LIN {X 0,Y 338.105,Z 590.455,A -85,B 0,C 180,E1 14436.471,E2 14436.471} C_VEL
LIN {X 0,Y 336.895,Z 591.514,A -85,B 0,C 180,E1 14436.227,E2 14436.227} C_VEL
LIN {X 0,Y 331.702,Z 598.648,A -85,B 0,C 180,E1 14435.239,E2 14435.239} C_VEL
LIN {X 0,Y 327.518,Z 602.639,A -85,B 0,C 180,E1 14434.334,E2 14434.334} C_VEL
LIN {X 0,Y 325.57,Z 603.97,A -85,B 0,C 180,E1 14433.877,E2 14433.877} C_VEL
LIN {X 0,Y 320.508,Z 612.012,A -85,B 0,C 180,E1 14432.822,E2 14432.822} C_VEL
LIN {X 0,Y 316.738,Z 616.286,A -85,B 0,C 180,E1 14431.922,E2 14431.922} C_VEL
LIN {X 0,Y 314.815,Z 617.214,A -85,B 0,C 180,E1 14431.391,E2 14431.391} C_VEL
LIN {X 0,Y 314.423,Z 617.302,A -85,B 0,C 180,E1 14431.251,E2 14431.251} C_VEL
LIN {X 0,Y 311.704,Z 638.432,A -85,B 0,C 180,E1 14428.545,E2 14428.545} C_VEL
LIN {X 0,Y 311.765,Z 644.155,A -85,B 0,C 180,E1 14428.291,E2 14428.291} C_VEL
LIN {X 0,Y 303.31,Z 754.586,A -85,B 0,C 180,E1 14423.992,E2 14423.992} C_VEL
LIN {X 0,Y 301.747,Z 787.034,A -85,B 0,C 180,E1 14422.515,E2 14422.515} C_VEL
LIN {X 0,Y 300.704,Z 803.184,A -85,B 0,C 180,E1 14421.454,E2 14421.454} C_VEL
LIN {X 0,Y 299.299,Z 819.779,A -85,B 0,C 180,E1 14419.987,E2 14419.987} C_VEL
LIN {X 0,Y 297.78,Z 834.708,A -85,B 0,C 180,E1 14418.298,E2 14418.298} C_VEL
LIN {X 0,Y 296.083,Z 849.627,A -85,B 0,C 180,E1 14416.177,E2 14416.177} C_VEL
LIN {X 0,Y 294.448,Z 863.222,A -85,B 0,C 180,E1 14413.751,E2 14413.751} C_VEL
LIN {X 0,Y 293.091,Z 874.714,A -85,B 0,C 180,E1 14411.213,E2 14411.213} C_VEL
LIN {X 0,Y 291.948,Z 885.373,A -85,B 0,C 180,E1 14408.27,E2 14408.27} C_VEL
LIN {X 0,Y 291.167,Z 894.27,A -85,B 0,C 180,E1 14405.123,E2 14405.123} C_VEL
LIN {X 0,Y 290.847,Z 900.711,A -85,B 0,C 180,E1 14402.167,E2 14402.167} C_VEL
LIN {X 0,Y 290.9,Z 906.041,A -85,B 0,C 180,E1 14398.819,E2 14398.819} C_VEL
LIN {X 0,Y 291.395,Z 909.402,A -85,B 0,C 180,E1 14395.474,E2 14395.474} C_VEL
LIN {X 0,Y 292.318,Z 910.935,A -85,B 0,C 180,E1 14392.334,E2 14392.334} C_VEL
LIN {X 0,Y 293.979,Z 910.74,A -85,B 0,C 180,E1 14388.822,E2 14388.822} C_VEL
LIN {X 0,Y 296.38,Z 908.513,A -85,B 0,C 180,E1 14385.344,E2 14385.344} C_VEL
LIN {X 0,Y 299.304,Z 904.667,A -85,B 0,C 180,E1 14382.193,E2 14382.193} C_VEL
LIN {X 0,Y 302.949,Z 899.041,A -85,B 0,C 180,E1 14379.118,E2 14379.118} C_VEL
LIN {X 0,Y 307.224,Z 891.662,A -85,B 0,C 180,E1 14376.2,E2 14376.2} C_VEL
LIN {X 0,Y 311.889,Z 882.811,A -85,B 0,C 180,E1 14373.538,E2 14373.538} C_VEL
LIN {X 0,Y 317.212,Z 871.822,A -85,B 0,C 180,E1 14370.961,E2 14370.961} C_VEL
LIN {X 0,Y 322.811,Z 859.287,A -85,B 0,C 180,E1 14368.644,E2 14368.644} C_VEL
LIN {X 0,Y 328.898,Z 844.76,A -85,B 0,C 180,E1 14366.512,E2 14366.512} C_VEL
LIN {X 0,Y 335.235,Z 828.569,A -85,B 0,C 180,E1 14364.647,E2 14364.647} C_VEL
LIN {X 0,Y 344.132,Z 807.464,A -85,B 0,C 180,E1 14362.715,E2 14362.715} C_VEL
LIN {X 0,Y 354.941,Z 783.665,A -85,B 0,C 180,E1 14360.98,E2 14360.98} C_VEL
LIN {X 0,Y 365.49,Z 758.939,A -85,B 0,C 180,E1 14359.583,E2 14359.583} C_VEL
LIN {X 0,Y 366.222,Z 757.158,A -85,B 0,C 180,E1 14359.481,E2 14359.481} C_VEL
LIN {X 0,Y 359.783,Z 774.746,A -85,B 0,C 180,E1 14358.984,E2 14358.984} C_VEL
LIN {X 0,Y 353.257,Z 791.701,A -85,B 0,C 180,E1 14358.23,E2 14358.23} C_VEL
LIN {X 0,Y 342.525,Z 818.157,A -85,B 0,C 180,E1 14356.624,E2 14356.624} C_VEL
LIN {X 0,Y 334.303,Z 838.121,A -85,B 0,C 180,E1 14355.081,E2 14355.081} C_VEL
LIN {X 0,Y 330.317,Z 857.082,A -85,B 0,C 180,E1 14353.883,E2 14353.883} C_VEL
LIN {X 0,Y 325.728,Z 875.895,A -85,B 0,C 180,E1 14352.361,E2 14352.361} C_VEL
LIN {X 0,Y 320.539,Z 894.611,A -85,B 0,C 180,E1 14350.454,E2 14350.454} C_VEL
LIN {X 0,Y 315.4,Z 911.334,A -85,B 0,C 180,E1 14348.35,E2 14348.35} C_VEL
LIN {X 0,Y 310.233,Z 927.162,A -85,B 0,C 180,E1 14345.915,E2 14345.915} C_VEL
LIN {X 0,Y 305.231,Z 941.839,A -85,B 0,C 180,E1 14343.166,E2 14343.166} C_VEL
LIN {X 0,Y 300.629,Z 955.074,A -85,B 0,C 180,E1 14340.147,E2 14340.147} C_VEL
LIN {X 0,Y 296.615,Z 966.984,A -85,B 0,C 180,E1 14336.854,E2 14336.854} C_VEL
LIN {X 0,Y 293.159,Z 978.066,A -85,B 0,C 180,E1 14333.094,E2 14333.094} C_VEL
LIN {X 0,Y 290.587,Z 987.507,A -85,B 0,C 180,E1 14329.081,E2 14329.081} C_VEL
LIN {X 0,Y 289.081,Z 994.669,A -85,B 0,C 180,E1 14325.207,E2 14325.207} C_VEL
LIN {X 0,Y 288.342,Z 1000.295,A -85,B 0,C 180,E1 14321.198,E2 14321.198} C_VEL
LIN {X 0,Y 288.162,Z 1003.977,A -85,B 0,C 180,E1 14317.377,E2 14317.377} C_VEL
LIN {X 0,Y 288.251,Z 1006.151,A -85,B 0,C 180,E1 14313.581,E2 14313.581} C_VEL
LIN {X 0,Y 288.329,Z 1006.883,A -85,B 0,C 180,E1 14310.001,E2 14310.001} C_VEL
LIN {X 0,Y 288.247,Z 1006.145,A -85,B 0,C 180,E1 14306.421,E2 14306.421} C_VEL
LIN {X 0,Y 288.144,Z 1003.964,A -85,B 0,C 180,E1 14302.625,E2 14302.625} C_VEL
LIN {X 0,Y 288.325,Z 1000.281,A -85,B 0,C 180,E1 14298.803,E2 14298.803} C_VEL
LIN {X 0,Y 289.07,Z 994.6,A -85,B 0,C 180,E1 14294.76,E2 14294.76} C_VEL
LIN {X 0,Y 290.554,Z 987.48,A -85,B 0,C 180,E1 14290.919,E2 14290.919} C_VEL
LIN {X 0,Y 292.964,Z 978.552,A -85,B 0,C 180,E1 14287.104,E2 14287.104} C_VEL
LIN {X 0,Y 296.275,Z 967.843,A -85,B 0,C 180,E1 14283.42,E2 14283.42} C_VEL
LIN {X 0,Y 300.323,Z 955.793,A -85,B 0,C 180,E1 14280.041,E2 14280.041} C_VEL
LIN {X 0,Y 304.862,Z 942.662,A -85,B 0,C 180,E1 14277.015,E2 14277.015} C_VEL
LIN {X 0,Y 309.992,Z 927.6,A -85,B 0,C 180,E1 14274.173,E2 14274.173} C_VEL
LIN {X 0,Y 315.053,Z 912.094,A -85,B 0,C 180,E1 14271.769,E2 14271.769} C_VEL
LIN {X 0,Y 320.25,Z 895.206,A -85,B 0,C 180,E1 14269.622,E2 14269.622} C_VEL
LIN {X 0,Y 325.17,Z 877.603,A -85,B 0,C 180,E1 14267.802,E2 14267.802} C_VEL
LIN {X 0,Y 329.756,Z 859.099,A -85,B 0,C 180,E1 14266.266,E2 14266.266} C_VEL
LIN {X 0,Y 333.969,Z 839.227,A -85,B 0,C 180,E1 14264.985,E2 14264.985} C_VEL
LIN {X 0,Y 337.417,Z 818.867,A -85,B 0,C 180,E1 14264.011,E2 14264.011} C_VEL
LIN {X 0,Y 339.946,Z 798.236,A -85,B 0,C 180,E1 14263.309,E2 14263.309} C_VEL
LIN {X 0,Y 341.701,Z 774.328,A -85,B 0,C 180,E1 14262.775,E2 14262.775} C_VEL
LIN {X 0,Y 344.693,Z 746.04,A -85,B 0,C 180,E1 14262.462,E2 14262.462} C_VEL
LIN {X 0,Y 348.273,Z 722.638,A -85,B 0,C 180,E1 14262.405,E2 14262.405} C_VEL
LIN {X 0,Y 349.346,Z 716.122,A -85,B 0,C 180,E1 14262.403,E2 14262.403} C_VEL
LIN {X 0,Y 343.198,Z 700.036,A -85,B 0,C 180,E1 14260.778,E2 14260.778} C_VEL
LIN {X 0,Y 338.934,Z 686.753,A -85,B 0,C 180,E1 14259.515,E2 14259.515} C_VEL
LIN {X 0,Y 337.267,Z 665.975,A -85,B 0,C 180,E1 14256.787,E2 14256.787} C_VEL
LIN {X 0,Y 338.08,Z 643.412,A -85,B 0,C 180,E1 14253.984,E2 14253.984} C_VEL
LIN {X 0,Y 341.699,Z 617.006,A -85,B 0,C 180,E1 14250.98,E2 14250.98} C_VEL
LIN {X 0,Y 346.458,Z 593.984,A -85,B 0,C 180,E1 14248.53,E2 14248.53} C_VEL
LIN {X 0,Y 338.453,Z 575.878,A -85,B 0,C 180,E1 14244.616,E2 14244.616} C_VEL
LIN {X 0,Y 330.252,Z 558.135,A -85,B 0,C 180,E1 14240.375,E2 14240.375} C_VEL
LIN {X 0,Y 322.963,Z 542.982,A -85,B 0,C 180,E1 14236.363,E2 14236.363} C_VEL
LIN {X 0,Y 316.245,Z 529.387,A -85,B 0,C 180,E1 14232.415,E2 14232.415} C_VEL
LIN {X 0,Y 309.793,Z 516.677,A -85,B 0,C 180,E1 14228.351,E2 14228.351} C_VEL
LIN {X 0,Y 304.602,Z 506.811,A -85,B 0,C 180,E1 14224.896,E2 14224.896} C_VEL
LIN {X 0,Y 301.925,Z 501.833,A -85,B 0,C 180,E1 14223.037,E2 14223.037} C_VEL
LIN {X 0,Y 299.876,Z 497.861,A -85,B 0,C 180,E1 14221.528,E2 14221.528} C_VEL
LIN {X 0,Y 297.644,Z 493.478,A -85,B 0,C 180,E1 14219.807,E2 14219.807} C_VEL
LIN {X 0,Y 295.15,Z 488.762,A -85,B 0,C 180,E1 14217.864,E2 14217.864} C_VEL
LIN {X 0,Y 293.163,Z 485.098,A -85,B 0,C 180,E1 14216.284,E2 14216.284} C_VEL
LIN {X 0,Y 292.668,Z 484.054,A -85,B 0,C 180,E1 14215.797,E2 14215.797} C_VEL
LIN {X 0,Y 295.376,Z 485.784,A -85,B 0,C 180,E1 14210.452,E2 14210.452} C_VEL
LIN {X 0,Y 296.859,Z 489.544,A -85,B 0,C 180,E1 14207.617,E2 14207.617} C_VEL
LIN {X 0,Y 299.685,Z 492.227,A -85,B 0,C 180,E1 14204.519,E2 14204.519} C_VEL
LIN {X 0,Y 301.439,Z 495.849,A -85,B 0,C 180,E1 14202.431,E2 14202.431} C_VEL
LIN {X 0,Y 303.501,Z 497.912,A -85,B 0,C 180,E1 14200.765,E2 14200.765} C_VEL
LIN {X 0,Y 305.517,Z 501.787,A -85,B 0,C 180,E1 14198.859,E2 14198.859} C_VEL
LIN {X 0,Y 307.211,Z 503.912,A -85,B 0,C 180,E1 14197.617,E2 14197.617} C_VEL
LIN {X 0,Y 309.597,Z 507.894,A -85,B 0,C 180,E1 14195.785,E2 14195.785} C_VEL
LIN {X 0,Y 310.833,Z 509.839,A -85,B 0,C 180,E1 14194.976,E2 14194.976} C_VEL
LIN {X 0,Y 315.313,Z 515.527,A -85,B 0,C 180,E1 14192.983,E2 14192.983} C_VEL
LIN {X 0,Y 322.031,Z 524.183,A -85,B 0,C 180,E1 14190.315,E2 14190.315} C_VEL
LIN {X 0,Y 329.717,Z 535.071,A -85,B 0,C 180,E1 14187.589,E2 14187.589} C_VEL
LIN {X 0,Y 338.579,Z 548.442,A -85,B 0,C 180,E1 14184.788,E2 14184.788} C_VEL
LIN {X 0,Y 347.19,Z 562.872,A -85,B 0,C 180,E1 14182.32,E2 14182.32} C_VEL
LIN {X 0,Y 352.785,Z 573.372,A -85,B 0,C 180,E1 14180.813,E2 14180.813} C_VEL
LIN {X 0,Y 342.08,Z 768.353,A -85,B 0,C 180,E1 14176.743,E2 14176.743} C_VEL
LIN {X 0,Y 340.044,Z 788.682,A -85,B 0,C 180,E1 14176.065,E2 14176.065} C_VEL
LIN {X 0,Y 337.064,Z 809.308,A -85,B 0,C 180,E1 14175.089,E2 14175.089} C_VEL
LIN {X 0,Y 333.401,Z 828.945,A -85,B 0,C 180,E1 14173.848,E2 14173.848} C_VEL
LIN {X 0,Y 329.276,Z 847.192,A -85,B 0,C 180,E1 14172.384,E2 14172.384} C_VEL
LIN {X 0,Y 324.469,Z 865.449,A -85,B 0,C 180,E1 14170.556,E2 14170.556} C_VEL
LIN {X 0,Y 319.337,Z 882.593,A -85,B 0,C 180,E1 14168.425,E2 14168.425} C_VEL
LIN {X 0,Y 314.214,Z 898.139,A -85,B 0,C 180,E1 14166.063,E2 14166.063} C_VEL
LIN {X 0,Y 309.078,Z 912.768,A -85,B 0,C 180,E1 14163.362,E2 14163.362} C_VEL
LIN {X 0,Y 304.251,Z 925.958,A -85,B 0,C 180,E1 14160.403,E2 14160.403} C_VEL
LIN {X 0,Y 299.884,Z 937.76,A -85,B 0,C 180,E1 14157.178,E2 14157.178} C_VEL
LIN {X 0,Y 296.107,Z 948.172,A -85,B 0,C 180,E1 14153.691,E2 14153.691} C_VEL
LIN {X 0,Y 292.892,Z 957.541,A -85,B 0,C 180,E1 14149.752,E2 14149.752} C_VEL
LIN {X 0,Y 290.646,Z 964.872,A -85,B 0,C 180,E1 14145.769,E2 14145.769} C_VEL
LIN {X 0,Y 289.234,Z 970.366,A -85,B 0,C 180,E1 14141.767,E2 14141.767} C_VEL
LIN {X 0,Y 288.495,Z 974.186,A -85,B 0,C 180,E1 14137.767,E2 14137.767} C_VEL
LIN {X 0,Y 288.2,Z 976.439,A -85,B 0,C 180,E1 14133.778,E2 14133.778} C_VEL
LIN {X 0,Y 288.153,Z 977.191,A -85,B 0,C 180,E1 14129.999,E2 14129.999} C_VEL
LIN {X 0,Y 288.196,Z 976.474,A -85,B 0,C 180,E1 14126.219,E2 14126.219} C_VEL
LIN {X 0,Y 288.491,Z 974.268,A -85,B 0,C 180,E1 14122.231,E2 14122.231} C_VEL
LIN {X 0,Y 289.216,Z 970.493,A -85,B 0,C 180,E1 14118.23,E2 14118.23} C_VEL
LIN {X 0,Y 290.613,Z 965.045,A -85,B 0,C 180,E1 14114.227,E2 14114.227} C_VEL
LIN {X 0,Y 292.838,Z 957.741,A -85,B 0,C 180,E1 14110.242,E2 14110.242} C_VEL
LIN {X 0,Y 295.849,Z 948.926,A -85,B 0,C 180,E1 14106.496,E2 14106.496} C_VEL
LIN {X 0,Y 299.563,Z 938.69,A -85,B 0,C 180,E1 14103.003,E2 14103.003} C_VEL
LIN {X 0,Y 303.878,Z 927.084,A -85,B 0,C 180,E1 14099.772,E2 14099.772} C_VEL
LIN {X 0,Y 308.641,Z 914.122,A -85,B 0,C 180,E1 14096.804,E2 14096.804} C_VEL
LIN {X 0,Y 313.738,Z 899.761,A -85,B 0,C 180,E1 14094.097,E2 14094.097} C_VEL
LIN {X 0,Y 319.007,Z 883.854,A -85,B 0,C 180,E1 14091.64,E2 14091.64} C_VEL
LIN {X 0,Y 320.725,Z 878.233,A -85,B 0,C 180,E1 14090.892,E2 14090.892} C_VEL
LIN {X 0,Y 321.773,Z 872.311,A -85,B 0,C 180,E1 14090.018,E2 14090.018} C_VEL
LIN {X 0,Y 321.585,Z 857.401,A -85,B 0,C 180,E1 14087.619,E2 14087.619} C_VEL
LIN {X 0,Y 322.577,Z 850.944,A -85,B 0,C 180,E1 14086.866,E2 14086.866} C_VEL
LIN {X 0,Y 327.274,Z 831.492,A -85,B 0,C 180,E1 14085.233,E2 14085.233} C_VEL
LIN {X 0,Y 331.162,Z 811.905,A -85,B 0,C 180,E1 14083.949,E2 14083.949} C_VEL
LIN {X 0,Y 334.256,Z 792.087,A -85,B 0,C 180,E1 14082.966,E2 14082.966} C_VEL
LIN {X 0,Y 336.537,Z 771.573,A -85,B 0,C 180,E1 14082.238,E2 14082.238} C_VEL
LIN {X 0,Y 338.982,Z 730.81,A -85,B 0,C 180,E1 14081.332,E2 14081.332} C_VEL
LIN {X 0,Y 346.754,Z 591.172,A -85,B 0,C 180,E1 14078.4,E2 14078.4} C_VEL
LIN {X 0,Y 341.098,Z 596.488,A -85,B 0,C 180,E1 14077.357,E2 14077.357} C_VEL
LIN {X 0,Y 338.973,Z 598.24,A -85,B 0,C 180,E1 14076.942,E2 14076.942} C_VEL
LIN {X 0,Y 333.543,Z 605.341,A -85,B 0,C 180,E1 14075.93,E2 14075.93} C_VEL
LIN {X 0,Y 328.773,Z 609.786,A -85,B 0,C 180,E1 14074.925,E2 14074.925} C_VEL
LIN {X 0,Y 327.374,Z 611,A -85,B 0,C 180,E1 14074.617,E2 14074.617} C_VEL
LIN {X 0,Y 322.039,Z 618.933,A -85,B 0,C 180,E1 14073.523,E2 14073.523} C_VEL
LIN {X 0,Y 317.705,Z 623.542,A -85,B 0,C 180,E1 14072.505,E2 14072.505} C_VEL
LIN {X 0,Y 315.69,Z 625.062,A -85,B 0,C 180,E1 14071.987,E2 14071.987} C_VEL
LIN {X 0,Y 310.632,Z 633.768,A -85,B 0,C 180,E1 14070.837,E2 14070.837} C_VEL
LIN {X 0,Y 306.71,Z 638.82,A -85,B 0,C 180,E1 14069.811,E2 14069.811} C_VEL
LIN {X 0,Y 304.863,Z 640.068,A -85,B 0,C 180,E1 14069.254,E2 14069.254} C_VEL
LIN {X 0,Y 304.63,Z 640.238,A -85,B 0,C 180,E1 14069.157,E2 14069.157} C_VEL
LIN {X 0,Y 304.475,Z 646.416,A -85,B 0,C 180,E1 14068.891,E2 14068.891} C_VEL
LIN {X 0,Y 296.163,Z 749.756,A -85,B 0,C 180,E1 14064.746,E2 14064.746} C_VEL
LIN {X 0,Y 294.087,Z 788.133,A -85,B 0,C 180,E1 14062.936,E2 14062.936} C_VEL
LIN {X 0,Y 292.895,Z 805.59,A -85,B 0,C 180,E1 14061.74,E2 14061.74} C_VEL
LIN {X 0,Y 291.393,Z 822.484,A -85,B 0,C 180,E1 14060.173,E2 14060.173} C_VEL
LIN {X 0,Y 289.719,Z 838.078,A -85,B 0,C 180,E1 14058.304,E2 14058.304} C_VEL
LIN {X 0,Y 288.073,Z 851.952,A -85,B 0,C 180,E1 14056.225,E2 14056.225} C_VEL
LIN {X 0,Y 286.42,Z 865.303,A -85,B 0,C 180,E1 14053.732,E2 14053.732} C_VEL
LIN {X 0,Y 285.049,Z 876.605,A -85,B 0,C 180,E1 14051.124,E2 14051.124} C_VEL
LIN {X 0,Y 283.986,Z 886.554,A -85,B 0,C 180,E1 14048.3,E2 14048.3} C_VEL
LIN {X 0,Y 283.201,Z 895.525,A -85,B 0,C 180,E1 14045.064,E2 14045.064} C_VEL
LIN {X 0,Y 282.894,Z 902.008,A -85,B 0,C 180,E1 14042.026,E2 14042.026} C_VEL
LIN {X 0,Y 282.989,Z 907.395,A -85,B 0,C 180,E1 14038.583,E2 14038.583} C_VEL
LIN {X 0,Y 283.56,Z 910.849,A -85,B 0,C 180,E1 14035.146,E2 14035.146} C_VEL
LIN {X 0,Y 284.592,Z 912.479,A -85,B 0,C 180,E1 14031.922,E2 14031.922} C_VEL
LIN {X 0,Y 286.415,Z 912.379,A -85,B 0,C 180,E1 14028.319,E2 14028.319} C_VEL
LIN {X 0,Y 288.878,Z 910.465,A -85,B 0,C 180,E1 14024.947,E2 14024.947} C_VEL
LIN {X 0,Y 292.097,Z 906.788,A -85,B 0,C 180,E1 14021.644,E2 14021.644} C_VEL
LIN {X 0,Y 295.88,Z 901.604,A -85,B 0,C 180,E1 14018.595,E2 14018.595} C_VEL
LIN {X 0,Y 300.729,Z 894.12,A -85,B 0,C 180,E1 14015.443,E2 14015.443} C_VEL
LIN {X 0,Y 306.074,Z 884.99,A -85,B 0,C 180,E1 14012.574,E2 14012.574} C_VEL
LIN {X 0,Y 311.856,Z 874.233,A -85,B 0,C 180,E1 14009.96,E2 14009.96} C_VEL
LIN {X 0,Y 318.274,Z 861.401,A -85,B 0,C 180,E1 14007.507,E2 14007.507} C_VEL
LIN {X 0,Y 325.112,Z 846.91,A -85,B 0,C 180,E1 14005.323,E2 14005.323} C_VEL
LIN {X 0,Y 332.308,Z 830.975,A -85,B 0,C 180,E1 14003.434,E2 14003.434} C_VEL
LIN {X 0,Y 342.206,Z 810.381,A -85,B 0,C 180,E1 14001.513,E2 14001.513} C_VEL
LIN {X 0,Y 353.925,Z 786.933,A -85,B 0,C 180,E1 13999.805,E2 13999.805} C_VEL
LIN {X 0,Y 341.598,Z 815.298,A -85,B 0,C 180,E1 13998.154,E2 13998.154} C_VEL
LIN {X 0,Y 331.581,Z 837.093,A -85,B 0,C 180,E1 13996.488,E2 13996.488} C_VEL
LIN {X 0,Y 326.37,Z 848.727,A -85,B 0,C 180,E1 13995.422,E2 13995.422} C_VEL
LIN {X 0,Y 321.853,Z 867.686,A -85,B 0,C 180,E1 13994.024,E2 13994.024} C_VEL
LIN {X 0,Y 316.918,Z 885.711,A -85,B 0,C 180,E1 13992.345,E2 13992.345} C_VEL
LIN {X 0,Y 311.504,Z 903.397,A -85,B 0,C 180,E1 13990.3,E2 13990.3} C_VEL
LIN {X 0,Y 305.913,Z 920.116,A -85,B 0,C 180,E1 13987.914,E2 13987.914} C_VEL
LIN {X 0,Y 300.747,Z 934.869,A -85,B 0,C 180,E1 13985.345,E2 13985.345} C_VEL
LIN {X 0,Y 295.362,Z 949.685,A -85,B 0,C 180,E1 13982.189,E2 13982.189} C_VEL
LIN {X 0,Y 290.692,Z 962.647,A -85,B 0,C 180,E1 13978.787,E2 13978.787} C_VEL
LIN {X 0,Y 286.823,Z 973.843,A -85,B 0,C 180,E1 13975.17,E2 13975.17} C_VEL
LIN {X 0,Y 283.918,Z 983.101,A -85,B 0,C 180,E1 13971.486,E2 13971.486} C_VEL
LIN {X 0,Y 281.792,Z 991.402,A -85,B 0,C 180,E1 13967.342,E2 13967.342} C_VEL
LIN {X 0,Y 280.618,Z 997.788,A -85,B 0,C 180,E1 13963.183,E2 13963.183} C_VEL
LIN {X 0,Y 280.199,Z 1002.226,A -85,B 0,C 180,E1 13959.242,E2 13959.242} C_VEL
LIN {X 0,Y 280.2,Z 1005.012,A -85,B 0,C 180,E1 13955.325,E2 13955.325} C_VEL
LIN {X 0,Y 280.316,Z 1006.314,A -85,B 0,C 180,E1 13951.432,E2 13951.432} C_VEL
LIN {X 0,Y 280.302,Z 1006.239,A -85,B 0,C 180,E1 13947.957,E2 13947.957} C_VEL
LIN {X 0,Y 280.189,Z 1004.765,A -85,B 0,C 180,E1 13944.267,E2 13944.267} C_VEL
LIN {X 0,Y 280.205,Z 1001.796,A -85,B 0,C 180,E1 13940.346,E2 13940.346} C_VEL
LIN {X 0,Y 280.712,Z 996.98,A -85,B 0,C 180,E1 13936.195,E2 13936.195} C_VEL
LIN {X 0,Y 282.02,Z 990.286,A -85,B 0,C 180,E1 13932.036,E2 13932.036} C_VEL
LIN {X 0,Y 284.166,Z 982.125,A -85,B 0,C 180,E1 13928.102,E2 13928.102} C_VEL
LIN {X 0,Y 287.344,Z 972.038,A -85,B 0,C 180,E1 13924.219,E2 13924.219} C_VEL
LIN {X 0,Y 291.38,Z 960.449,A -85,B 0,C 180,E1 13920.615,E2 13920.615} C_VEL
LIN {X 0,Y 295.796,Z 948.237,A -85,B 0,C 180,E1 13917.491,E2 13917.491} C_VEL
LIN {X 0,Y 301.059,Z 933.777,A -85,B 0,C 180,E1 13914.457,E2 13914.457} C_VEL
LIN {X 0,Y 306.645,Z 917.765,A -85,B 0,C 180,E1 13911.72,E2 13911.72} C_VEL
LIN {X 0,Y 312.268,Z 900.704,A -85,B 0,C 180,E1 13909.363,E2 13909.363} C_VEL
LIN {X 0,Y 317.555,Z 883.096,A -85,B 0,C 180,E1 13907.395,E2 13907.395} C_VEL
LIN {X 0,Y 322.455,Z 864.747,A -85,B 0,C 180,E1 13905.748,E2 13905.748} C_VEL
LIN {X 0,Y 327.088,Z 844.606,A -85,B 0,C 180,E1 13904.333,E2 13904.333} C_VEL
LIN {X 0,Y 330.916,Z 824.384,A -85,B 0,C 180,E1 13903.267,E2 13903.267} C_VEL
LIN {X 0,Y 333.828,Z 804.122,A -85,B 0,C 180,E1 13902.494,E2 13902.494} C_VEL
LIN {X 0,Y 335.696,Z 782.554,A -85,B 0,C 180,E1 13901.923,E2 13901.923} C_VEL
LIN {X 0,Y 338.017,Z 756.825,A -85,B 0,C 180,E1 13901.559,E2 13901.559} C_VEL
LIN {X 0,Y 341.555,Z 730.296,A -85,B 0,C 180,E1 13901.405,E2 13901.405} C_VEL
LIN {X 0,Y 343.552,Z 718.12,A -85,B 0,C 180,E1 13901.405,E2 13901.405} C_VEL
LIN {X 0,Y 338.467,Z 704.5,A -85,B 0,C 180,E1 13899.993,E2 13899.993} C_VEL
LIN {X 0,Y 334.162,Z 690.716,A -85,B 0,C 180,E1 13898.654,E2 13898.654} C_VEL
LIN {X 0,Y 330.754,Z 677.82,A -85,B 0,C 180,E1 13897.472,E2 13897.472} C_VEL
LIN {X 0,Y 330.542,Z 655.887,A -85,B 0,C 180,E1 13894.638,E2 13894.638} C_VEL
LIN {X 0,Y 333.093,Z 630.866,A -85,B 0,C 180,E1 13891.623,E2 13891.623} C_VEL
LIN {X 0,Y 339,Z 600.919,A -85,B 0,C 180,E1 13888.35,E2 13888.35} C_VEL
LIN {X 0,Y 339.708,Z 597.396,A -85,B 0,C 180,E1 13887.959,E2 13887.959} C_VEL
LIN {X 0,Y 331.773,Z 579.454,A -85,B 0,C 180,E1 13884.007,E2 13884.007} C_VEL
LIN {X 0,Y 323.613,Z 561.719,A -85,B 0,C 180,E1 13879.68,E2 13879.68} C_VEL
LIN {X 0,Y 316.63,Z 547.214,A -85,B 0,C 180,E1 13875.758,E2 13875.758} C_VEL
LIN {X 0,Y 310.532,Z 534.705,A -85,B 0,C 180,E1 13872.08,E2 13872.08} C_VEL
LIN {X 0,Y 304.052,Z 521.904,A -85,B 0,C 180,E1 13867.938,E2 13867.938} C_VEL
LIN {X 0,Y 299.144,Z 512.458,A -85,B 0,C 180,E1 13864.601,E2 13864.601} C_VEL
LIN {X 0,Y 294.678,Z 503.883,A -85,B 0,C 180,E1 13861.361,E2 13861.361} C_VEL
LIN {X 0,Y 291.974,Z 498.82,A -85,B 0,C 180,E1 13859.316,E2 13859.316} C_VEL
LIN {X 0,Y 289.601,Z 494.32,A -85,B 0,C 180,E1 13857.427,E2 13857.427} C_VEL
LIN {X 0,Y 289.077,Z 493.536,A -85,B 0,C 180,E1 13857.026,E2 13857.026} C_VEL
LIN {X 0,Y 290.16,Z 491.712,A -85,B 0,C 180,E1 13855.454,E2 13855.454} C_VEL
LIN {X 0,Y 292.456,Z 493.411,A -85,B 0,C 180,E1 13850.554,E2 13850.554} C_VEL
LIN {X 0,Y 294.168,Z 497.263,A -85,B 0,C 180,E1 13847.436,E2 13847.436} C_VEL
LIN {X 0,Y 296.458,Z 499.205,A -85,B 0,C 180,E1 13844.948,E2 13844.948} C_VEL
LIN {X 0,Y 298.283,Z 503.117,A -85,B 0,C 180,E1 13842.642,E2 13842.642} C_VEL
LIN {X 0,Y 300.209,Z 505.352,A -85,B 0,C 180,E1 13840.95,E2 13840.95} C_VEL
LIN {X 0,Y 302.429,Z 509.28,A -85,B 0,C 180,E1 13838.877,E2 13838.877} C_VEL
LIN {X 0,Y 303.79,Z 510.952,A -85,B 0,C 180,E1 13837.963,E2 13837.963} C_VEL
LIN {X 0,Y 307.344,Z 515.372,A -85,B 0,C 180,E1 13836.107,E2 13836.107} C_VEL
LIN {X 0,Y 313.061,Z 522.818,A -85,B 0,C 180,E1 13833.44,E2 13833.44} C_VEL
LIN {X 0,Y 319.551,Z 531.401,A -85,B 0,C 180,E1 13830.783,E2 13830.783} C_VEL
LIN {X 0,Y 327.112,Z 542.313,A -85,B 0,C 180,E1 13828.024,E2 13828.024} C_VEL
LIN {X 0,Y 335.839,Z 555.837,A -85,B 0,C 180,E1 13825.188,E2 13825.188} C_VEL
LIN {X 0,Y 343.944,Z 569.808,A -85,B 0,C 180,E1 13822.795,E2 13822.795} C_VEL
LIN {X 0,Y 347.604,Z 576.808,A -85,B 0,C 180,E1 13821.769,E2 13821.769} C_VEL
LIN {X 0,Y 336.644,Z 768.776,A -85,B 0,C 180,E1 13817.731,E2 13817.731} C_VEL
LIN {X 0,Y 334.531,Z 789.158,A -85,B 0,C 180,E1 13817.047,E2 13817.047} C_VEL
LIN {X 0,Y 331.454,Z 809.731,A -85,B 0,C 180,E1 13816.067,E2 13816.067} C_VEL
LIN {X 0,Y 327.667,Z 829.336,A -85,B 0,C 180,E1 13814.819,E2 13814.819} C_VEL
LIN {X 0,Y 323.39,Z 847.59,A -85,B 0,C 180,E1 13813.343,E2 13813.343} C_VEL
LIN {X 0,Y 318.398,Z 865.853,A -85,B 0,C 180,E1 13811.497,E2 13811.497} C_VEL
LIN {X 0,Y 313.06,Z 883,A -85,B 0,C 180,E1 13809.343,E2 13809.343} C_VEL
LIN {X 0,Y 307.65,Z 898.739,A -85,B 0,C 180,E1 13806.917,E2 13806.917} C_VEL
LIN {X 0,Y 302.348,Z 913.181,A -85,B 0,C 180,E1 13804.206,E2 13804.206} C_VEL
LIN {X 0,Y 297.279,Z 926.373,A -85,B 0,C 180,E1 13801.194,E2 13801.194} C_VEL
LIN {X 0,Y 292.684,Z 938.176,A -85,B 0,C 180,E1 13797.904,E2 13797.904} C_VEL
LIN {X 0,Y 288.688,Z 948.589,A -85,B 0,C 180,E1 13794.339,E2 13794.339} C_VEL
LIN {X 0,Y 285.269,Z 957.958,A -85,B 0,C 180,E1 13790.302,E2 13790.302} C_VEL
LIN {X 0,Y 282.864,Z 965.29,A -85,B 0,C 180,E1 13786.214,E2 13786.214} C_VEL
LIN {X 0,Y 281.341,Z 970.782,A -85,B 0,C 180,E1 13782.102,E2 13782.102} C_VEL
LIN {X 0,Y 280.537,Z 974.6,A -85,B 0,C 180,E1 13777.989,E2 13777.989} C_VEL
LIN {X 0,Y 280.217,Z 976.851,A -85,B 0,C 180,E1 13773.886,E2 13773.886} C_VEL
LIN {X 0,Y 280.163,Z 977.603,A -85,B 0,C 180,E1 13769.999,E2 13769.999} C_VEL
LIN {X 0,Y 280.213,Z 976.886,A -85,B 0,C 180,E1 13766.111,E2 13766.111} C_VEL
LIN {X 0,Y 280.531,Z 974.682,A -85,B 0,C 180,E1 13762.009,E2 13762.009} C_VEL
LIN {X 0,Y 281.322,Z 970.907,A -85,B 0,C 180,E1 13757.894,E2 13757.894} C_VEL
LIN {X 0,Y 282.829,Z 965.46,A -85,B 0,C 180,E1 13753.782,E2 13753.782} C_VEL
LIN {X 0,Y 285.213,Z 958.156,A -85,B 0,C 180,E1 13749.691,E2 13749.691} C_VEL
LIN {X 0,Y 288.416,Z 949.34,A -85,B 0,C 180,E1 13745.852,E2 13745.852} C_VEL
LIN {X 0,Y 292.346,Z 939.102,A -85,B 0,C 180,E1 13742.28,E2 13742.28} C_VEL
LIN {X 0,Y 296.889,Z 927.494,A -85,B 0,C 180,E1 13738.983,E2 13738.983} C_VEL
LIN {X 0,Y 301.895,Z 914.53,A -85,B 0,C 180,E1 13735.963,E2 13735.963} C_VEL
LIN {X 0,Y 307.222,Z 900.165,A -85,B 0,C 180,E1 13733.213,E2 13733.213} C_VEL
LIN {X 0,Y 312.874,Z 883.798,A -85,B 0,C 180,E1 13730.658,E2 13730.658} C_VEL
LIN {X 0,Y 318.255,Z 866.549,A -85,B 0,C 180,E1 13728.478,E2 13728.478} C_VEL
LIN {X 0,Y 322.577,Z 850.944,A -85,B 0,C 180,E1 13726.866,E2 13726.866} C_VEL
LIN {X 0,Y 323.572,Z 844.413,A -85,B 0,C 180,E1 13726.144,E2 13726.144} C_VEL
LIN {X 0,Y 323.23,Z 828.017,A -85,B 0,C 180,E1 13724.078,E2 13724.078} C_VEL
LIN {X 0,Y 323.951,Z 821.097,A -85,B 0,C 180,E1 13723.476,E2 13723.476} C_VEL
LIN {X 0,Y 327.606,Z 800.708,A -85,B 0,C 180,E1 13722.322,E2 13722.322} C_VEL
LIN {X 0,Y 330.319,Z 780.399,A -85,B 0,C 180,E1 13721.484,E2 13721.484} C_VEL
LIN {X 0,Y 332.147,Z 759.221,A -85,B 0,C 180,E1 13720.898,E2 13720.898} C_VEL
LIN {X 0,Y 341.004,Z 605.06,A -85,B 0,C 180,E1 13717.629,E2 13717.629} C_VEL
LIN {X 0,Y 335.209,Z 612.268,A -85,B 0,C 180,E1 13716.571,E2 13716.571} C_VEL
LIN {X 0,Y 329.908,Z 617.04,A -85,B 0,C 180,E1 13715.478,E2 13715.478} C_VEL
LIN {X 0,Y 323.622,Z 625.817,A -85,B 0,C 180,E1 13714.216,E2 13714.216} C_VEL
LIN {X 0,Y 318.852,Z 630.681,A -85,B 0,C 180,E1 13713.122,E2 13713.122} C_VEL
LIN {X 0,Y 317.43,Z 632.017,A -85,B 0,C 180,E1 13712.778,E2 13712.778} C_VEL
LIN {X 0,Y 312.098,Z 640.643,A -85,B 0,C 180,E1 13711.588,E2 13711.588} C_VEL
LIN {X 0,Y 307.836,Z 645.832,A -85,B 0,C 180,E1 13710.498,E2 13710.498} C_VEL
LIN {X 0,Y 307.18,Z 646.678,A -85,B 0,C 180,E1 13710.327,E2 13710.327} C_VEL
LIN {X 0,Y 301.287,Z 670.598,A -85,B 0,C 180,E1 13709.499,E2 13709.499} C_VEL
LIN {X 0,Y 296.93,Z 685.296,A -85,B 0,C 180,E1 13708.703,E2 13708.703} C_VEL
LIN {X 0,Y 294.585,Z 691.14,A -85,B 0,C 180,E1 13708.15,E2 13708.15} C_VEL
LIN {X 0,Y 293.534,Z 692.236,A -85,B 0,C 180,E1 13707.818,E2 13707.818} C_VEL
LIN {X 0,Y 287.488,Z 768.614,A -85,B 0,C 180,E1 13704.428,E2 13704.428} C_VEL
LIN {X 0,Y 286.217,Z 792.991,A -85,B 0,C 180,E1 13703.149,E2 13703.149} C_VEL
LIN {X 0,Y 284.893,Z 810.241,A -85,B 0,C 180,E1 13701.84,E2 13701.84} C_VEL
LIN {X 0,Y 283.346,Z 826.198,A -85,B 0,C 180,E1 13700.232,E2 13700.232} C_VEL
LIN {X 0,Y 281.564,Z 841.939,A -85,B 0,C 180,E1 13698.21,E2 13698.21} C_VEL
LIN {X 0,Y 279.698,Z 856.968,A -85,B 0,C 180,E1 13695.765,E2 13695.765} C_VEL
LIN {X 0,Y 278.147,Z 869.166,A -85,B 0,C 180,E1 13693.301,E2 13693.301} C_VEL
LIN {X 0,Y 276.754,Z 880.819,A -85,B 0,C 180,E1 13690.407,E2 13690.407} C_VEL
LIN {X 0,Y 275.659,Z 891.351,A -85,B 0,C 180,E1 13687.084,E2 13687.084} C_VEL
LIN {X 0,Y 275.063,Z 899.53,A -85,B 0,C 180,E1 13683.752,E2 13683.752} C_VEL
LIN {X 0,Y 274.938,Z 905.758,A -85,B 0,C 180,E1 13680.417,E2 13680.417} C_VEL
LIN {X 0,Y 275.288,Z 910.437,A -85,B 0,C 180,E1 13676.877,E2 13676.877} C_VEL
LIN {X 0,Y 276.165,Z 913.227,A -85,B 0,C 180,E1 13673.347,E2 13673.347} C_VEL
LIN {X 0,Y 277.668,Z 914.261,A -85,B 0,C 180,E1 13669.838,E2 13669.838} C_VEL
LIN {X 0,Y 280.049,Z 913.453,A -85,B 0,C 180,E1 13666.16,E2 13666.16} C_VEL
LIN {X 0,Y 283.312,Z 910.699,A -85,B 0,C 180,E1 13662.544,E2 13662.544} C_VEL
LIN {X 0,Y 287.775,Z 905.594,A -85,B 0,C 180,E1 13658.818,E2 13658.818} C_VEL
LIN {X 0,Y 293.013,Z 898.529,A -85,B 0,C 180,E1 13655.399,E2 13655.399} C_VEL
LIN {X 0,Y 298.521,Z 890.295,A -85,B 0,C 180,E1 13652.47,E2 13652.47} C_VEL
LIN {X 0,Y 304.845,Z 880.001,A -85,B 0,C 180,E1 13649.662,E2 13649.662} C_VEL
LIN {X 0,Y 311.571,Z 868.266,A -85,B 0,C 180,E1 13647.158,E2 13647.158} C_VEL
LIN {X 0,Y 319.158,Z 854.204,A -85,B 0,C 180,E1 13644.8,E2 13644.8} C_VEL
LIN {X 0,Y 327.205,Z 838.762,A -85,B 0,C 180,E1 13642.769,E2 13642.769} C_VEL
LIN {X 0,Y 336.91,Z 820.434,A -85,B 0,C 180,E1 13640.903,E2 13640.903} C_VEL
LIN {X 0,Y 343.283,Z 808.945,A -85,B 0,C 180,E1 13639.933,E2 13639.933} C_VEL
LIN {X 0,Y 332.387,Z 831.126,A -85,B 0,C 180,E1 13638.377,E2 13638.377} C_VEL
LIN {X 0,Y 321.879,Z 851.849,A -85,B 0,C 180,E1 13636.497,E2 13636.497} C_VEL
LIN {X 0,Y 318.09,Z 859.544,A -85,B 0,C 180,E1 13635.665,E2 13635.665} C_VEL
LIN {X 0,Y 312.684,Z 879.604,A -85,B 0,C 180,E1 13633.941,E2 13633.941} C_VEL
LIN {X 0,Y 307.165,Z 897.5,A -85,B 0,C 180,E1 13631.986,E2 13631.986} C_VEL
LIN {X 0,Y 301.581,Z 913.846,A -85,B 0,C 180,E1 13629.784,E2 13629.784} C_VEL
LIN {X 0,Y 295.753,Z 929.924,A -85,B 0,C 180,E1 13627.119,E2 13627.119} C_VEL
LIN {X 0,Y 290.242,Z 944.474,A -85,B 0,C 180,E1 13624.162,E2 13624.162} C_VEL
LIN {X 0,Y 285.358,Z 957.242,A -85,B 0,C 180,E1 13621.003,E2 13621.003} C_VEL
LIN {X 0,Y 280.849,Z 969.326,A -85,B 0,C 180,E1 13617.34,E2 13617.34} C_VEL
LIN {X 0,Y 277.226,Z 979.851,A -85,B 0,C 180,E1 13613.375,E2 13613.375} C_VEL
LIN {X 0,Y 274.553,Z 988.745,A -85,B 0,C 180,E1 13609.134,E2 13609.134} C_VEL
LIN {X 0,Y 272.968,Z 995.658,A -85,B 0,C 180,E1 13604.858,E2 13604.858} C_VEL
LIN {X 0,Y 272.3,Z 1000.537,A -85,B 0,C 180,E1 13600.794,E2 13600.794} C_VEL
LIN {X 0,Y 272.193,Z 1004.004,A -85,B 0,C 180,E1 13596.54,E2 13596.54} C_VEL
LIN {X 0,Y 272.29,Z 1005.681,A -85,B 0,C 180,E1 13592.737,E2 13592.737} C_VEL
LIN {X 0,Y 272.331,Z 1005.949,A -85,B 0,C 180,E1 13588.949,E2 13588.949} C_VEL
LIN {X 0,Y 272.218,Z 1004.942,A -85,B 0,C 180,E1 13585.155,E2 13585.155} C_VEL
LIN {X 0,Y 272.18,Z 1002.3,A -85,B 0,C 180,E1 13581.126,E2 13581.126} C_VEL
LIN {X 0,Y 272.577,Z 997.879,A -85,B 0,C 180,E1 13576.856,E2 13576.856} C_VEL
LIN {X 0,Y 273.772,Z 991.685,A -85,B 0,C 180,E1 13572.575,E2 13572.575} C_VEL
LIN {X 0,Y 275.828,Z 984.053,A -85,B 0,C 180,E1 13568.525,E2 13568.525} C_VEL
LIN {X 0,Y 278.944,Z 974.536,A -85,B 0,C 180,E1 13564.525,E2 13564.525} C_VEL
LIN {X 0,Y 283.187,Z 962.851,A -85,B 0,C 180,E1 13560.61,E2 13560.61} C_VEL
LIN {X 0,Y 288.045,Z 950.018,A -85,B 0,C 180,E1 13557.143,E2 13557.143} C_VEL
LIN {X 0,Y 293.296,Z 936.233,A -85,B 0,C 180,E1 13554.103,E2 13554.103} C_VEL
LIN {X 0,Y 299.028,Z 920.708,A -85,B 0,C 180,E1 13551.299,E2 13551.299} C_VEL
LIN {X 0,Y 305.029,Z 903.52,A -85,B 0,C 180,E1 13548.788,E2 13548.788} C_VEL
LIN {X 0,Y 310.646,Z 885.947,A -85,B 0,C 180,E1 13546.721,E2 13546.721} C_VEL
LIN {X 0,Y 315.652,Z 868.472,A -85,B 0,C 180,E1 13545.061,E2 13545.061} C_VEL
LIN {X 0,Y 320.417,Z 849.287,A -85,B 0,C 180,E1 13543.619,E2 13543.619} C_VEL
LIN {X 0,Y 324.591,Z 828.93,A -85,B 0,C 180,E1 13542.462,E2 13542.462} C_VEL
LIN {X 0,Y 327.808,Z 808.742,A -85,B 0,C 180,E1 13541.629,E2 13541.629} C_VEL
LIN {X 0,Y 329.97,Z 787.868,A -85,B 0,C 180,E1 13541.019,E2 13541.019} C_VEL
LIN {X 0,Y 331.982,Z 763.663,A -85,B 0,C 180,E1 13540.603,E2 13540.603} C_VEL
LIN {X 0,Y 335.802,Z 733.241,A -85,B 0,C 180,E1 13540.384,E2 13540.384} C_VEL
LIN {X 0,Y 337.812,Z 720.281,A -85,B 0,C 180,E1 13540.368,E2 13540.368} C_VEL
LIN {X 0,Y 330.68,Z 699.292,A -85,B 0,C 180,E1 13538.194,E2 13538.194} C_VEL
LIN {X 0,Y 326.105,Z 681.524,A -85,B 0,C 180,E1 13536.536,E2 13536.536} C_VEL
LIN {X 0,Y 323.435,Z 669.067,A -85,B 0,C 180,E1 13535.438,E2 13535.438} C_VEL
LIN {X 0,Y 324.645,Z 646.262,A -85,B 0,C 180,E1 13532.545,E2 13532.545} C_VEL
LIN {X 0,Y 328.817,Z 619.429,A -85,B 0,C 180,E1 13529.405,E2 13529.405} C_VEL
LIN {X 0,Y 332.89,Z 600.698,A -85,B 0,C 180,E1 13527.357,E2 13527.357} C_VEL
LIN {X 0,Y 325.406,Z 583.754,A -85,B 0,C 180,E1 13523.543,E2 13523.543} C_VEL
LIN {X 0,Y 317.288,Z 565.906,A -85,B 0,C 180,E1 13519.131,E2 13519.131} C_VEL
LIN {X 0,Y 309.727,Z 550.111,A -85,B 0,C 180,E1 13514.775,E2 13514.775} C_VEL
LIN {X 0,Y 303.082,Z 536.488,A -85,B 0,C 180,E1 13510.646,E2 13510.646} C_VEL
LIN {X 0,Y 296.395,Z 523.269,A -85,B 0,C 180,E1 13506.197,E2 13506.197} C_VEL
LIN {X 0,Y 291.526,Z 513.957,A -85,B 0,C 180,E1 13502.752,E2 13502.752} C_VEL
LIN {X 0,Y 286.878,Z 504.987,A -85,B 0,C 180,E1 13499.201,E2 13499.201} C_VEL
LIN {X 0,Y 285.786,Z 502.828,A -85,B 0,C 180,E1 13498.195,E2 13498.195} C_VEL
LIN {X 0,Y 287.676,Z 499.359,A -85,B 0,C 180,E1 13495.215,E2 13495.215} C_VEL
LIN {X 0,Y 289.722,Z 500.948,A -85,B 0,C 180,E1 13490.75,E2 13490.75} C_VEL
LIN {X 0,Y 291.319,Z 504.744,A -85,B 0,C 180,E1 13487.512,E2 13487.512} C_VEL
LIN {X 0,Y 293.32,Z 506.579,A -85,B 0,C 180,E1 13485.187,E2 13485.187} C_VEL
LIN {X 0,Y 295.317,Z 510.632,A -85,B 0,C 180,E1 13482.666,E2 13482.666} C_VEL
LIN {X 0,Y 297.156,Z 512.546,A -85,B 0,C 180,E1 13481.307,E2 13481.307} C_VEL
LIN {X 0,Y 300.575,Z 516.935,A -85,B 0,C 180,E1 13479.149,E2 13479.149} C_VEL
LIN {X 0,Y 301.997,Z 518.607,A -85,B 0,C 180,E1 13478.336,E2 13478.336} C_VEL
LIN {X 0,Y 306.617,Z 524.535,A -85,B 0,C 180,E1 13475.893,E2 13475.893} C_VEL
LIN {X 0,Y 311.113,Z 530.51,A -85,B 0,C 180,E1 13473.775,E2 13473.775} C_VEL
LIN {X 0,Y 317.094,Z 538.609,A -85,B 0,C 180,E1 13471.258,E2 13471.258} C_VEL
LIN {X 0,Y 325.209,Z 550.499,A -85,B 0,C 180,E1 13468.23,E2 13468.23} C_VEL
LIN {X 0,Y 334.441,Z 565.469,A -85,B 0,C 180,E1 13465.178,E2 13465.178} C_VEL
LIN {X 0,Y 342.52,Z 580.098,A -85,B 0,C 180,E1 13462.76,E2 13462.76} C_VEL
LIN {X 0,Y 331.312,Z 769.205,A -85,B 0,C 180,E1 13458.752,E2 13458.752} C_VEL
LIN {X 0,Y 329.134,Z 789.521,A -85,B 0,C 180,E1 13458.066,E2 13458.066} C_VEL
LIN {X 0,Y 325.942,Z 810.163,A -85,B 0,C 180,E1 13457.077,E2 13457.077} C_VEL
LIN {X 0,Y 322.03,Z 829.728,A -85,B 0,C 180,E1 13455.824,E2 13455.824} C_VEL
LIN {X 0,Y 317.597,Z 847.989,A -85,B 0,C 180,E1 13454.338,E2 13454.338} C_VEL
LIN {X 0,Y 312.416,Z 866.257,A -85,B 0,C 180,E1 13452.475,E2 13452.475} C_VEL
LIN {X 0,Y 306.979,Z 883.062,A -85,B 0,C 180,E1 13450.345,E2 13450.345} C_VEL
LIN {X 0,Y 301.296,Z 898.961,A -85,B 0,C 180,E1 13447.873,E2 13447.873} C_VEL
LIN {X 0,Y 295.661,Z 913.656,A -85,B 0,C 180,E1 13445.076,E2 13445.076} C_VEL
LIN {X 0,Y 290.369,Z 926.789,A -85,B 0,C 180,E1 13442.023,E2 13442.023} C_VEL
LIN {X 0,Y 285.534,Z 938.593,A -85,B 0,C 180,E1 13438.667,E2 13438.667} C_VEL
LIN {X 0,Y 281.257,Z 949.128,A -85,B 0,C 180,E1 13434.971,E2 13434.971} C_VEL
LIN {X 0,Y 277.672,Z 958.376,A -85,B 0,C 180,E1 13430.883,E2 13430.883} C_VEL
LIN {X 0,Y 275.098,Z 965.707,A -85,B 0,C 180,E1 13426.685,E2 13426.685} C_VEL
LIN {X 0,Y 273.458,Z 971.198,A -85,B 0,C 180,E1 13422.457,E2 13422.457} C_VEL
LIN {X 0,Y 272.584,Z 975.014,A -85,B 0,C 180,E1 13418.224,E2 13418.224} C_VEL
LIN {X 0,Y 272.234,Z 977.263,A -85,B 0,C 180,E1 13414,E2 13414} C_VEL
LIN {X 0,Y 272.174,Z 978.014,A -85,B 0,C 180,E1 13409.999,E2 13409.999} C_VEL
LIN {X 0,Y 272.231,Z 977.298,A -85,B 0,C 180,E1 13405.997,E2 13405.997} C_VEL
LIN {X 0,Y 272.575,Z 975.095,A -85,B 0,C 180,E1 13401.774,E2 13401.774} C_VEL
LIN {X 0,Y 273.379,Z 971.566,A -85,B 0,C 180,E1 13397.752,E2 13397.752} C_VEL
LIN {X 0,Y 274.959,Z 966.188,A -85,B 0,C 180,E1 13393.521,E2 13393.521} C_VEL
LIN {X 0,Y 277.459,Z 958.962,A -85,B 0,C 180,E1 13389.318,E2 13389.318} C_VEL
LIN {X 0,Y 280.815,Z 950.253,A -85,B 0,C 180,E1 13385.38,E2 13385.38} C_VEL
LIN {X 0,Y 284.924,Z 940.133,A -85,B 0,C 180,E1 13381.721,E2 13381.721} C_VEL
LIN {X 0,Y 289.961,Z 927.905,A -85,B 0,C 180,E1 13378.157,E2 13378.157} C_VEL
LIN {X 0,Y 295.354,Z 914.588,A -85,B 0,C 180,E1 13375.009,E2 13375.009} C_VEL
LIN {X 0,Y 300.784,Z 900.569,A -85,B 0,C 180,E1 13372.29,E2 13372.29} C_VEL
LIN {X 0,Y 306.576,Z 884.493,A -85,B 0,C 180,E1 13369.744,E2 13369.744} C_VEL
LIN {X 0,Y 312.042,Z 867.662,A -85,B 0,C 180,E1 13367.584,E2 13367.584} C_VEL
LIN {X 0,Y 316.964,Z 850.583,A -85,B 0,C 180,E1 13365.8,E2 13365.8} C_VEL
LIN {X 0,Y 321.629,Z 831.871,A -85,B 0,C 180,E1 13364.227,E2 13364.227} C_VEL
LIN {X 0,Y 323.951,Z 821.097,A -85,B 0,C 180,E1 13363.476,E2 13363.476} C_VEL
LIN {X 0,Y 324.697,Z 814.062,A -85,B 0,C 180,E1 13362.909,E2 13362.909} C_VEL
LIN {X 0,Y 323.721,Z 796.475,A -85,B 0,C 180,E1 13361.198,E2 13361.198} C_VEL
LIN {X 0,Y 324.037,Z 789.172,A -85,B 0,C 180,E1 13360.747,E2 13360.747} C_VEL
LIN {X 0,Y 326.313,Z 768.041,A -85,B 0,C 180,E1 13360.048,E2 13360.048} C_VEL
LIN {X 0,Y 335.241,Z 620.845,A -85,B 0,C 180,E1 13356.881,E2 13356.881} C_VEL
LIN {X 0,Y 331.43,Z 624.382,A -85,B 0,C 180,E1 13356.115,E2 13356.115} C_VEL
LIN {X 0,Y 325.497,Z 632.397,A -85,B 0,C 180,E1 13354.952,E2 13354.952} C_VEL
LIN {X 0,Y 320.338,Z 637.579,A -85,B 0,C 180,E1 13353.805,E2 13353.805} C_VEL
LIN {X 0,Y 319.132,Z 639.061,A -85,B 0,C 180,E1 13353.537,E2 13353.537} C_VEL
LIN {X 0,Y 313.594,Z 647.516,A -85,B 0,C 180,E1 13352.325,E2 13352.325} C_VEL
LIN {X 0,Y 310.167,Z 651.943,A -85,B 0,C 180,E1 13351.496,E2 13351.496} C_VEL
LIN {X 0,Y 304.219,Z 675.229,A -85,B 0,C 180,E1 13350.681,E2 13350.681} C_VEL
LIN {X 0,Y 299.867,Z 689.311,A -85,B 0,C 180,E1 13349.911,E2 13349.911} C_VEL
LIN {X 0,Y 297.106,Z 695.971,A -85,B 0,C 180,E1 13349.291,E2 13349.291} C_VEL
LIN {X 0,Y 296.052,Z 698.047,A -85,B 0,C 180,E1 13349.024,E2 13349.024} C_VEL
LIN {X 0,Y 290.223,Z 722.088,A -85,B 0,C 180,E1 13348.13,E2 13348.13} C_VEL
LIN {X 0,Y 285.53,Z 738.516,A -85,B 0,C 180,E1 13347.204,E2 13347.204} C_VEL
LIN {X 0,Y 282.875,Z 745.651,A -85,B 0,C 180,E1 13346.532,E2 13346.532} C_VEL
LIN {X 0,Y 281.889,Z 747.103,A -85,B 0,C 180,E1 13346.206,E2 13346.206} C_VEL
LIN {X 0,Y 281.444,Z 747.266,A -85,B 0,C 180,E1 13346.013,E2 13346.013} C_VEL
LIN {X 0,Y 278.836,Z 789.509,A -85,B 0,C 180,E1 13343.879,E2 13343.879} C_VEL
LIN {X 0,Y 277.476,Z 807.748,A -85,B 0,C 180,E1 13342.55,E2 13342.55} C_VEL
LIN {X 0,Y 275.778,Z 825.255,A -85,B 0,C 180,E1 13340.813,E2 13340.813} C_VEL
LIN {X 0,Y 274.001,Z 840.657,A -85,B 0,C 180,E1 13338.842,E2 13338.842} C_VEL
LIN {X 0,Y 272.266,Z 854.492,A -85,B 0,C 180,E1 13336.646,E2 13336.646} C_VEL
LIN {X 0,Y 270.468,Z 868.307,A -85,B 0,C 180,E1 13333.904,E2 13333.904} C_VEL
LIN {X 0,Y 268.966,Z 880.284,A -85,B 0,C 180,E1 13330.929,E2 13330.929} C_VEL
LIN {X 0,Y 267.912,Z 890.026,A -85,B 0,C 180,E1 13327.937,E2 13327.937} C_VEL
LIN {X 0,Y 267.203,Z 898.887,A -85,B 0,C 180,E1 13324.507,E2 13324.507} C_VEL
LIN {X 0,Y 266.978,Z 905.613,A -85,B 0,C 180,E1 13321.073,E2 13321.073} C_VEL
LIN {X 0,Y 267.231,Z 910.6,A -85,B 0,C 180,E1 13317.642,E2 13317.642} C_VEL
LIN {X 0,Y 268.106,Z 914.202,A -85,B 0,C 180,E1 13313.792,E2 13313.792} C_VEL
LIN {X 0,Y 269.596,Z 915.745,A -85,B 0,C 180,E1 13310.178,E2 13310.178} C_VEL
LIN {X 0,Y 271.836,Z 915.59,A -85,B 0,C 180,E1 13306.602,E2 13306.602} C_VEL
LIN {X 0,Y 275.113,Z 913.556,A -85,B 0,C 180,E1 13302.88,E2 13302.88} C_VEL
LIN {X 0,Y 279.351,Z 909.587,A -85,B 0,C 180,E1 13299.247,E2 13299.247} C_VEL
LIN {X 0,Y 284.615,Z 903.565,A -85,B 0,C 180,E1 13295.731,E2 13295.731} C_VEL
LIN {X 0,Y 290.932,Z 895.378,A -85,B 0,C 180,E1 13292.357,E2 13292.357} C_VEL
LIN {X 0,Y 297.443,Z 886.121,A -85,B 0,C 180,E1 13289.497,E2 13289.497} C_VEL
LIN {X 0,Y 304.836,Z 874.786,A -85,B 0,C 180,E1 13286.787,E2 13286.787} C_VEL
LIN {X 0,Y 313.222,Z 861.21,A -85,B 0,C 180,E1 13284.256,E2 13284.256} C_VEL
LIN {X 0,Y 322.154,Z 846.217,A -85,B 0,C 180,E1 13282.083,E2 13282.083} C_VEL
LIN {X 0,Y 332.049,Z 829.42,A -85,B 0,C 180,E1 13280.218,E2 13280.218} C_VEL
LIN {X 0,Y 332.889,Z 828.082,A -85,B 0,C 180,E1 13280.057,E2 13280.057} C_VEL
LIN {X 0,Y 321.507,Z 848.789,A -85,B 0,C 180,E1 13278.279,E2 13278.279} C_VEL
LIN {X 0,Y 310.687,Z 867.822,A -85,B 0,C 180,E1 13276.129,E2 13276.129} C_VEL
LIN {X 0,Y 309.229,Z 870.961,A -85,B 0,C 180,E1 13275.743,E2 13275.743} C_VEL
LIN {X 0,Y 304.348,Z 887.358,A -85,B 0,C 180,E1 13274.146,E2 13274.146} C_VEL
LIN {X 0,Y 298.548,Z 904.604,A -85,B 0,C 180,E1 13272.054,E2 13272.054} C_VEL
LIN {X 0,Y 292.583,Z 920.822,A -85,B 0,C 180,E1 13269.63,E2 13269.63} C_VEL
LIN {X 0,Y 286.367,Z 936.851,A -85,B 0,C 180,E1 13266.66,E2 13266.66} C_VEL
LIN {X 0,Y 280.787,Z 950.696,A -85,B 0,C 180,E1 13263.502,E2 13263.502} C_VEL
LIN {X 0,Y 275.816,Z 963.138,A -85,B 0,C 180,E1 13260.019,E2 13260.019} C_VEL
LIN {X 0,Y 271.565,Z 974.165,A -85,B 0,C 180,E1 13256.221,E2 13256.221} C_VEL
LIN {X 0,Y 268.212,Z 983.669,A -85,B 0,C 180,E1 13252.119,E2 13252.119} C_VEL
LIN {X 0,Y 265.991,Z 991.29,A -85,B 0,C 180,E1 13247.954,E2 13247.954} C_VEL
LIN {X 0,Y 264.675,Z 997.479,A -85,B 0,C 180,E1 13243.547,E2 13243.547} C_VEL
LIN {X 0,Y 264.202,Z 1001.898,A -85,B 0,C 180,E1 13239.147,E2 13239.147} C_VEL
LIN {X 0,Y 264.223,Z 1004.538,A -85,B 0,C 180,E1 13234.994,E2 13234.994} C_VEL
LIN {X 0,Y 264.341,Z 1005.539,A -85,B 0,C 180,E1 13231.085,E2 13231.085} C_VEL
LIN {X 0,Y 264.294,Z 1005.263,A -85,B 0,C 180,E1 13227.182,E2 13227.182} C_VEL
LIN {X 0,Y 264.174,Z 1003.578,A -85,B 0,C 180,E1 13223.263,E2 13223.263} C_VEL
LIN {X 0,Y 264.296,Z 1000.317,A -85,B 0,C 180,E1 13219.098,E2 13219.098} C_VEL
LIN {X 0,Y 265.052,Z 995.216,A -85,B 0,C 180,E1 13214.69,E2 13214.69} C_VEL
LIN {X 0,Y 266.656,Z 988.703,A -85,B 0,C 180,E1 13210.507,E2 13210.507} C_VEL
LIN {X 0,Y 269.464,Z 979.868,A -85,B 0,C 180,E1 13206.145,E2 13206.145} C_VEL
LIN {X 0,Y 273.272,Z 969.435,A -85,B 0,C 180,E1 13202.075,E2 13202.075} C_VEL
LIN {X 0,Y 277.692,Z 958.179,A -85,B 0,C 180,E1 13198.529,E2 13198.529} C_VEL
LIN {X 0,Y 283.073,Z 944.827,A -85,B 0,C 180,E1 13195.097,E2 13195.097} C_VEL
LIN {X 0,Y 288.998,Z 929.912,A -85,B 0,C 180,E1 13191.989,E2 13191.989} C_VEL
LIN {X 0,Y 294.846,Z 914.527,A -85,B 0,C 180,E1 13189.377,E2 13189.377} C_VEL
LIN {X 0,Y 300.845,Z 897.669,A -85,B 0,C 180,E1 13187.055,E2 13187.055} C_VEL
LIN {X 0,Y 306.779,Z 879.145,A -85,B 0,C 180,E1 13185.011,E2 13185.011} C_VEL
LIN {X 0,Y 312.127,Z 860.04,A -85,B 0,C 180,E1 13183.352,E2 13183.352} C_VEL
LIN {X 0,Y 316.607,Z 841.271,A -85,B 0,C 180,E1 13182.087,E2 13182.087} C_VEL
LIN {X 0,Y 320.514,Z 821.27,A -85,B 0,C 180,E1 13181.067,E2 13181.067} C_VEL
LIN {X 0,Y 323.624,Z 799.592,A -85,B 0,C 180,E1 13180.278,E2 13180.278} C_VEL
LIN {X 0,Y 325.674,Z 775.738,A -85,B 0,C 180,E1 13179.71,E2 13179.71} C_VEL
LIN {X 0,Y 328.665,Z 747.707,A -85,B 0,C 180,E1 13179.399,E2 13179.399} C_VEL
LIN {X 0,Y 332.214,Z 723.424,A -85,B 0,C 180,E1 13179.333,E2 13179.333} C_VEL
LIN {X 0,Y 332.138,Z 722.212,A -85,B 0,C 180,E1 13179.277,E2 13179.277} C_VEL
LIN {X 0,Y 325.334,Z 700.617,A -85,B 0,C 180,E1 13177.04,E2 13177.04} C_VEL
LIN {X 0,Y 320.062,Z 678.857,A -85,B 0,C 180,E1 13174.963,E2 13174.963} C_VEL
LIN {X 0,Y 316.872,Z 660.467,A -85,B 0,C 180,E1 13173.409,E2 13173.409} C_VEL
LIN {X 0,Y 319.633,Z 635.364,A -85,B 0,C 180,E1 13170.305,E2 13170.305} C_VEL
LIN {X 0,Y 325.678,Z 606.374,A -85,B 0,C 180,E1 13167.024,E2 13167.024} C_VEL
LIN {X 0,Y 326.173,Z 604.218,A -85,B 0,C 180,E1 13166.783,E2 13166.783} C_VEL
LIN {X 0,Y 318.664,Z 587.239,A -85,B 0,C 180,E1 13162.896,E2 13162.896} C_VEL
LIN {X 0,Y 310.894,Z 570.008,A -85,B 0,C 180,E1 13158.565,E2 13158.565} C_VEL
LIN {X 0,Y 303.372,Z 554.148,A -85,B 0,C 180,E1 13154.116,E2 13154.116} C_VEL
LIN {X 0,Y 296.711,Z 540.595,A -85,B 0,C 180,E1 13149.896,E2 13149.896} C_VEL
LIN {X 0,Y 290.597,Z 528.4,A -85,B 0,C 180,E1 13145.726,E2 13145.726} C_VEL
LIN {X 0,Y 285.715,Z 519.006,A -85,B 0,C 180,E1 13142.206,E2 13142.206} C_VEL
LIN {X 0,Y 282.48,Z 512.519,A -85,B 0,C 180,E1 13139.594,E2 13139.594} C_VEL
LIN {X 0,Y 284.389,Z 508.065,A -85,B 0,C 180,E1 13135.968,E2 13135.968} C_VEL
LIN {X 0,Y 285.118,Z 506.985,A -85,B 0,C 180,E1 13134.97,E2 13134.97} C_VEL
LIN {X 0,Y 286.862,Z 508.382,A -85,B 0,C 180,E1 13130.976,E2 13130.976} C_VEL
LIN {X 0,Y 288.494,Z 512.232,A -85,B 0,C 180,E1 13127.591,E2 13127.591} C_VEL
LIN {X 0,Y 290.8,Z 514.299,A -85,B 0,C 180,E1 13125.361,E2 13125.361} C_VEL
LIN {X 0,Y 293.946,Z 518.549,A -85,B 0,C 180,E1 13122.786,E2 13122.786} C_VEL
LIN {X 0,Y 295.551,Z 520.268,A -85,B 0,C 180,E1 13121.662,E2 13121.662} C_VEL
LIN {X 0,Y 299.149,Z 524.776,A -85,B 0,C 180,E1 13119.352,E2 13119.352} C_VEL
LIN {X 0,Y 304.498,Z 531.81,A -85,B 0,C 180,E1 13116.384,E2 13116.384} C_VEL
LIN {X 0,Y 310.812,Z 540.254,A -85,B 0,C 180,E1 13113.387,E2 13113.387} C_VEL
LIN {X 0,Y 318.182,Z 551.021,A -85,B 0,C 180,E1 13110.334,E2 13110.334} C_VEL
LIN {X 0,Y 325.49,Z 562.451,A -85,B 0,C 180,E1 13107.658,E2 13107.658} C_VEL
LIN {X 0,Y 333.689,Z 576.449,A -85,B 0,C 180,E1 13104.957,E2 13104.957} C_VEL
LIN {X 0,Y 337.523,Z 584.007,A -85,B 0,C 180,E1 13103.762,E2 13103.762} C_VEL
LIN {X 0,Y 326.088,Z 769.635,A -85,B 0,C 180,E1 13099.805,E2 13099.805} C_VEL
LIN {X 0,Y 323.829,Z 789.998,A -85,B 0,C 180,E1 13099.114,E2 13099.114} C_VEL
LIN {X 0,Y 320.535,Z 810.596,A -85,B 0,C 180,E1 13098.122,E2 13098.122} C_VEL
LIN {X 0,Y 316.497,Z 830.12,A -85,B 0,C 180,E1 13096.865,E2 13096.865} C_VEL
LIN {X 0,Y 311.905,Z 848.388,A -85,B 0,C 180,E1 13095.368,E2 13095.368} C_VEL
LIN {X 0,Y 306.529,Z 866.661,A -85,B 0,C 180,E1 13093.491,E2 13093.491} C_VEL
LIN {X 0,Y 300.779,Z 883.761,A -85,B 0,C 180,E1 13091.299,E2 13091.299} C_VEL
LIN {X 0,Y 294.958,Z 899.372,A -85,B 0,C 180,E1 13088.837,E2 13088.837} C_VEL
LIN {X 0,Y 289.095,Z 914.008,A -85,B 0,C 180,E1 13086.011,E2 13086.011} C_VEL
LIN {X 0,Y 283.526,Z 927.204,A -85,B 0,C 180,E1 13082.892,E2 13082.892} C_VEL
LIN {X 0,Y 278.437,Z 939.01,A -85,B 0,C 180,E1 13079.468,E2 13079.468} C_VEL
LIN {X 0,Y 273.97,Z 949.425,A -85,B 0,C 180,E1 13075.739,E2 13075.739} C_VEL
LIN {X 0,Y 270.271,Z 958.369,A -85,B 0,C 180,E1 13071.711,E2 13071.711} C_VEL
LIN {X 0,Y 267.461,Z 965.783,A -85,B 0,C 180,E1 13067.4,E2 13067.4} C_VEL
LIN {X 0,Y 265.65,Z 971.37,A -85,B 0,C 180,E1 13063.05,E2 13063.05} C_VEL
LIN {X 0,Y 264.669,Z 975.276,A -85,B 0,C 180,E1 13058.69,E2 13058.69} C_VEL
LIN {X 0,Y 264.277,Z 977.547,A -85,B 0,C 180,E1 13054.556,E2 13054.556} C_VEL
LIN {X 0,Y 264.177,Z 978.383,A -85,B 0,C 180,E1 13050.433,E2 13050.433} C_VEL
LIN {X 0,Y 264.227,Z 977.839,A -85,B 0,C 180,E1 13046.31,E2 13046.31} C_VEL
LIN {X 0,Y 264.57,Z 975.813,A -85,B 0,C 180,E1 13041.961,E2 13041.961} C_VEL
LIN {X 0,Y 265.437,Z 972.224,A -85,B 0,C 180,E1 13037.6,E2 13037.6} C_VEL
LIN {X 0,Y 267.2,Z 966.603,A -85,B 0,C 180,E1 13033.029,E2 13033.029} C_VEL
LIN {X 0,Y 269.881,Z 959.377,A -85,B 0,C 180,E1 13028.71,E2 13028.71} C_VEL
LIN {X 0,Y 273.45,Z 950.668,A -85,B 0,C 180,E1 13024.67,E2 13024.67} C_VEL
LIN {X 0,Y 277.798,Z 940.546,A -85,B 0,C 180,E1 13020.928,E2 13020.928} C_VEL
LIN {X 0,Y 283.099,Z 928.316,A -85,B 0,C 180,E1 13017.29,E2 13017.29} C_VEL
LIN {X 0,Y 288.617,Z 915.335,A -85,B 0,C 180,E1 13014.16,E2 13014.16} C_VEL
LIN {X 0,Y 294.428,Z 900.973,A -85,B 0,C 180,E1 13011.327,E2 13011.327} C_VEL
LIN {X 0,Y 300.406,Z 885.054,A -85,B 0,C 180,E1 13008.774,E2 13008.774} C_VEL
LIN {X 0,Y 306.147,Z 868.057,A -85,B 0,C 180,E1 13006.568,E2 13006.568} C_VEL
LIN {X 0,Y 311.253,Z 850.972,A -85,B 0,C 180,E1 13004.769,E2 13004.769} C_VEL
LIN {X 0,Y 316.088,Z 832.249,A -85,B 0,C 180,E1 13003.186,E2 13003.186} C_VEL
LIN {X 0,Y 320.282,Z 812.489,A -85,B 0,C 180,E1 13001.878,E2 13001.878} C_VEL
LIN {X 0,Y 323.58,Z 792.64,A -85,B 0,C 180,E1 13000.887,E2 13000.887} C_VEL
LIN {X 0,Y 324.037,Z 789.172,A -85,B 0,C 180,E1 13000.747,E2 13000.747} C_VEL
LIN {X 0,Y 324.331,Z 781.773,A -85,B 0,C 180,E1 13000.327,E2 13000.327} C_VEL
LIN {X 0,Y 322.285,Z 763.301,A -85,B 0,C 180,E1 12998.967,E2 12998.967} C_VEL
LIN {X 0,Y 322.146,Z 755.753,A -85,B 0,C 180,E1 12998.659,E2 12998.659} C_VEL
LIN {X 0,Y 329.56,Z 636.415,A -85,B 0,C 180,E1 12996.105,E2 12996.105} C_VEL
LIN {X 0,Y 323.576,Z 642.974,A -85,B 0,C 180,E1 12994.866,E2 12994.866} C_VEL
LIN {X 0,Y 321.368,Z 645.249,A -85,B 0,C 180,E1 12994.381,E2 12994.381} C_VEL
LIN {X 0,Y 315.355,Z 654.09,A -85,B 0,C 180,E1 12993.102,E2 12993.102} C_VEL
LIN {X 0,Y 313.352,Z 656.827,A -85,B 0,C 180,E1 12992.647,E2 12992.647} C_VEL
LIN {X 0,Y 307.287,Z 679.772,A -85,B 0,C 180,E1 12991.839,E2 12991.839} C_VEL
LIN {X 0,Y 302.863,Z 693.509,A -85,B 0,C 180,E1 12991.081,E2 12991.081} C_VEL
LIN {X 0,Y 299.667,Z 700.929,A -85,B 0,C 180,E1 12990.392,E2 12990.392} C_VEL
LIN {X 0,Y 298.987,Z 702.915,A -85,B 0,C 180,E1 12990.261,E2 12990.261} C_VEL
LIN {X 0,Y 292.975,Z 726.847,A -85,B 0,C 180,E1 12989.366,E2 12989.366} C_VEL
LIN {X 0,Y 288.189,Z 742.88,A -85,B 0,C 180,E1 12988.451,E2 12988.451} C_VEL
LIN {X 0,Y 285.235,Z 750.452,A -85,B 0,C 180,E1 12987.733,E2 12987.733} C_VEL
LIN {X 0,Y 283.704,Z 753.451,A -85,B 0,C 180,E1 12987.297,E2 12987.297} C_VEL
LIN {X 0,Y 279.189,Z 771.201,A -85,B 0,C 180,E1 12986.537,E2 12986.537} C_VEL
LIN {X 0,Y 275.917,Z 780.633,A -85,B 0,C 180,E1 12985.906,E2 12985.906} C_VEL
LIN {X 0,Y 273.274,Z 786.016,A -85,B 0,C 180,E1 12985.259,E2 12985.259} C_VEL
LIN {X 0,Y 271.89,Z 787.63,A -85,B 0,C 180,E1 12984.786,E2 12984.786} C_VEL
LIN {X 0,Y 271.347,Z 787.712,A -85,B 0,C 180,E1 12984.512,E2 12984.512} C_VEL
LIN {X 0,Y 270.13,Z 804.525,A -85,B 0,C 180,E1 12983.332,E2 12983.332} C_VEL
LIN {X 0,Y 268.545,Z 821.361,A -85,B 0,C 180,E1 12981.745,E2 12981.745} C_VEL
LIN {X 0,Y 266.719,Z 837.276,A -85,B 0,C 180,E1 12979.788,E2 12979.788} C_VEL
LIN {X 0,Y 264.885,Z 851.597,A -85,B 0,C 180,E1 12977.577,E2 12977.577} C_VEL
LIN {X 0,Y 263.007,Z 865.734,A -85,B 0,C 180,E1 12974.869,E2 12974.869} C_VEL
LIN {X 0,Y 261.298,Z 878.921,A -85,B 0,C 180,E1 12971.701,E2 12971.701} C_VEL
LIN {X 0,Y 260.065,Z 889.809,A -85,B 0,C 180,E1 12968.401,E2 12968.401} C_VEL
LIN {X 0,Y 259.31,Z 898.473,A -85,B 0,C 180,E1 12965.088,E2 12965.088} C_VEL
LIN {X 0,Y 259.024,Z 905.726,A -85,B 0,C 180,E1 12961.549,E2 12961.549} C_VEL
LIN {X 0,Y 259.265,Z 911.36,A -85,B 0,C 180,E1 12957.79,E2 12957.79} C_VEL
LIN {X 0,Y 260.099,Z 915.143,A -85,B 0,C 180,E1 12954.043,E2 12954.043} C_VEL
LIN {X 0,Y 261.622,Z 917.184,A -85,B 0,C 180,E1 12950.32,E2 12950.32} C_VEL
LIN {X 0,Y 264.075,Z 917.416,A -85,B 0,C 180,E1 12946.424,E2 12946.424} C_VEL
LIN {X 0,Y 267.513,Z 915.777,A -85,B 0,C 180,E1 12942.602,E2 12942.602} C_VEL
LIN {X 0,Y 271.683,Z 912.503,A -85,B 0,C 180,E1 12939.085,E2 12939.085} C_VEL
LIN {X 0,Y 276.813,Z 907.51,A -85,B 0,C 180,E1 12935.684,E2 12935.684} C_VEL
LIN {X 0,Y 283.299,Z 900.213,A -85,B 0,C 180,E1 12932.234,E2 12932.234} C_VEL
LIN {X 0,Y 290.433,Z 891.317,A -85,B 0,C 180,E1 12929.139,E2 12929.139} C_VEL
LIN {X 0,Y 298.597,Z 880.341,A -85,B 0,C 180,E1 12926.231,E2 12926.231} C_VEL
LIN {X 0,Y 307.297,Z 867.942,A -85,B 0,C 180,E1 12923.689,E2 12923.689} C_VEL
LIN {X 0,Y 317.154,Z 853.389,A -85,B 0,C 180,E1 12921.376,E2 12921.376} C_VEL
LIN {X 0,Y 323.09,Z 844.414,A -85,B 0,C 180,E1 12920.199,E2 12920.199} C_VEL
LIN {X 0,Y 312.227,Z 861.906,A -85,B 0,C 180,E1 12918.397,E2 12918.397} C_VEL
LIN {X 0,Y 301.831,Z 878.15,A -85,B 0,C 180,E1 12916.234,E2 12916.234} C_VEL
LIN {X 0,Y 300.399,Z 881.267,A -85,B 0,C 180,E1 12915.832,E2 12915.832} C_VEL
LIN {X 0,Y 294.508,Z 898.832,A -85,B 0,C 180,E1 12913.836,E2 12913.836} C_VEL
LIN {X 0,Y 288.066,Z 916.083,A -85,B 0,C 180,E1 12911.394,E2 12911.394} C_VEL
LIN {X 0,Y 281.618,Z 932.171,A -85,B 0,C 180,E1 12908.544,E2 12908.544} C_VEL
LIN {X 0,Y 275.705,Z 946.211,A -85,B 0,C 180,E1 12905.469,E2 12905.469} C_VEL
LIN {X 0,Y 270.399,Z 958.644,A -85,B 0,C 180,E1 12902.138,E2 12902.138} C_VEL
LIN {X 0,Y 265.325,Z 970.826,A -85,B 0,C 180,E1 12898.104,E2 12898.104} C_VEL
LIN {X 0,Y 261.455,Z 980.9,A -85,B 0,C 180,E1 12893.915,E2 12893.915} C_VEL
LIN {X 0,Y 258.724,Z 989.048,A -85,B 0,C 180,E1 12889.648,E2 12889.648} C_VEL
LIN {X 0,Y 257.009,Z 995.738,A -85,B 0,C 180,E1 12885.11,E2 12885.11} C_VEL
LIN {X 0,Y 256.281,Z 1000.595,A -85,B 0,C 180,E1 12880.533,E2 12880.533} C_VEL
LIN {X 0,Y 256.211,Z 1003.534,A -85,B 0,C 180,E1 12876.274,E2 12876.274} C_VEL
LIN {X 0,Y 256.325,Z 1005.005,A -85,B 0,C 180,E1 12872.237,E2 12872.237} C_VEL
LIN {X 0,Y 256.347,Z 1005.101,A -85,B 0,C 180,E1 12868.66,E2 12868.66} C_VEL
LIN {X 0,Y 256.213,Z 1003.997,A -85,B 0,C 180,E1 12864.627,E2 12864.627} C_VEL
LIN {X 0,Y 256.199,Z 1001.466,A -85,B 0,C 180,E1 12860.567,E2 12860.567} C_VEL
LIN {X 0,Y 256.723,Z 997.039,A -85,B 0,C 180,E1 12856.028,E2 12856.028} C_VEL
LIN {X 0,Y 258.167,Z 990.84,A -85,B 0,C 180,E1 12851.485,E2 12851.485} C_VEL
LIN {X 0,Y 260.576,Z 983.205,A -85,B 0,C 180,E1 12847.199,E2 12847.199} C_VEL
LIN {X 0,Y 264.146,Z 973.688,A -85,B 0,C 180,E1 12842.986,E2 12842.986} C_VEL
LIN {X 0,Y 268.943,Z 962.005,A -85,B 0,C 180,E1 12838.886,E2 12838.886} C_VEL
LIN {X 0,Y 274.249,Z 949.415,A -85,B 0,C 180,E1 12835.339,E2 12835.339} C_VEL
LIN {X 0,Y 279.766,Z 936.332,A -85,B 0,C 180,E1 12832.329,E2 12832.329} C_VEL
LIN {X 0,Y 286.203,Z 920.436,A -85,B 0,C 180,E1 12829.343,E2 12829.343} C_VEL
LIN {X 0,Y 292.468,Z 904.04,A -85,B 0,C 180,E1 12826.865,E2 12826.865} C_VEL
LIN {X 0,Y 298.498,Z 886.761,A -85,B 0,C 180,E1 12824.757,E2 12824.757} C_VEL
LIN {X 0,Y 304.2,Z 868.39,A -85,B 0,C 180,E1 12822.965,E2 12822.965} C_VEL
LIN {X 0,Y 309.496,Z 848.5,A -85,B 0,C 180,E1 12821.454,E2 12821.454} C_VEL
LIN {X 0,Y 313.951,Z 828.165,A -85,B 0,C 180,E1 12820.294,E2 12820.294} C_VEL
LIN {X 0,Y 317.376,Z 807.925,A -85,B 0,C 180,E1 12819.457,E2 12819.457} C_VEL
LIN {X 0,Y 319.675,Z 787.013,A -85,B 0,C 180,E1 12818.841,E2 12818.841} C_VEL
LIN {X 0,Y 321.938,Z 761.821,A -85,B 0,C 180,E1 12818.427,E2 12818.427} C_VEL
LIN {X 0,Y 325.832,Z 731.513,A -85,B 0,C 180,E1 12818.237,E2 12818.237} C_VEL
LIN {X 0,Y 326.835,Z 724.693,A -85,B 0,C 180,E1 12818.223,E2 12818.223} C_VEL
LIN {X 0,Y 320.656,Z 704.023,A -85,B 0,C 180,E1 12816.054,E2 12816.054} C_VEL
LIN {X 0,Y 315.709,Z 682.819,A -85,B 0,C 180,E1 12813.985,E2 12813.985} C_VEL
LIN {X 0,Y 312.533,Z 663.62,A -85,B 0,C 180,E1 12812.327,E2 12812.327} C_VEL
LIN {X 0,Y 310.967,Z 651.733,A -85,B 0,C 180,E1 12811.364,E2 12811.364} C_VEL
LIN {X 0,Y 315.236,Z 625.136,A -85,B 0,C 180,E1 12808.147,E2 12808.147} C_VEL
LIN {X 0,Y 319.302,Z 607.435,A -85,B 0,C 180,E1 12806.151,E2 12806.151} C_VEL
LIN {X 0,Y 311.633,Z 589.902,A -85,B 0,C 180,E1 12802.048,E2 12802.048} C_VEL
LIN {X 0,Y 303.882,Z 572.787,A -85,B 0,C 180,E1 12797.62,E2 12797.62} C_VEL
LIN {X 0,Y 295.834,Z 555.724,A -85,B 0,C 180,E1 12792.69,E2 12792.69} C_VEL
LIN {X 0,Y 289.21,Z 542.311,A -85,B 0,C 180,E1 12788.349,E2 12788.349} C_VEL
LIN {X 0,Y 283.502,Z 530.683,A -85,B 0,C 180,E1 12784.247,E2 12784.247} C_VEL
LIN {X 0,Y 280.573,Z 525.118,A -85,B 0,C 180,E1 12782.042,E2 12782.042} C_VEL
LIN {X 0,Y 281.118,Z 519.334,A -85,B 0,C 180,E1 12778.573,E2 12778.573} C_VEL
LIN {X 0,Y 282.68,Z 514.638,A -85,B 0,C 180,E1 12774.825,E2 12774.825} C_VEL
LIN {X 0,Y 284.622,Z 516.023,A -85,B 0,C 180,E1 12771.21,E2 12771.21} C_VEL
LIN {X 0,Y 287.066,Z 519.931,A -85,B 0,C 180,E1 12767.937,E2 12767.937} C_VEL
LIN {X 0,Y 289.386,Z 522.05,A -85,B 0,C 180,E1 12765.697,E2 12765.697} C_VEL
LIN {X 0,Y 292.594,Z 526.359,A -85,B 0,C 180,E1 12763.012,E2 12763.012} C_VEL
LIN {X 0,Y 293.96,Z 527.97,A -85,B 0,C 180,E1 12762.02,E2 12762.02} C_VEL
LIN {X 0,Y 298.381,Z 533.738,A -85,B 0,C 180,E1 12759.143,E2 12759.143} C_VEL
LIN {X 0,Y 302.484,Z 539.209,A -85,B 0,C 180,E1 12756.836,E2 12756.836} C_VEL
LIN {X 0,Y 308.481,Z 547.433,A -85,B 0,C 180,E1 12753.896,E2 12753.896} C_VEL
LIN {X 0,Y 315.6,Z 558.067,A -85,B 0,C 180,E1 12750.85,E2 12750.85} C_VEL
LIN {X 0,Y 322.929,Z 569.817,A -85,B 0,C 180,E1 12748.083,E2 12748.083} C_VEL
LIN {X 0,Y 330.941,Z 583.995,A -85,B 0,C 180,E1 12745.363,E2 12745.363} C_VEL
LIN {X 0,Y 332.639,Z 587.65,A -85,B 0,C 180,E1 12744.802,E2 12744.802} C_VEL
LIN {X 0,Y 320.978,Z 770.061,A -85,B 0,C 180,E1 12740.893,E2 12740.893} C_VEL
LIN {X 0,Y 318.667,Z 790.251,A -85,B 0,C 180,E1 12740.206,E2 12740.206} C_VEL
LIN {X 0,Y 315.241,Z 811.022,A -85,B 0,C 180,E1 12739.203,E2 12739.203} C_VEL
LIN {X 0,Y 311.072,Z 830.513,A -85,B 0,C 180,E1 12737.942,E2 12737.942} C_VEL
LIN {X 0,Y 306.318,Z 848.787,A -85,B 0,C 180,E1 12736.437,E2 12736.437} C_VEL
LIN {X 0,Y 300.742,Z 867.065,A -85,B 0,C 180,E1 12734.546,E2 12734.546} C_VEL
LIN {X 0,Y 294.667,Z 884.459,A -85,B 0,C 180,E1 12732.293,E2 12732.293} C_VEL
LIN {X 0,Y 288.497,Z 900.325,A -85,B 0,C 180,E1 12729.748,E2 12729.748} C_VEL
LIN {X 0,Y 282.583,Z 914.421,A -85,B 0,C 180,E1 12726.977,E2 12726.977} C_VEL
LIN {X 0,Y 276.749,Z 927.628,A -85,B 0,C 180,E1 12723.802,E2 12723.802} C_VEL
LIN {X 0,Y 271.398,Z 939.427,A -85,B 0,C 180,E1 12720.312,E2 12720.312} C_VEL
LIN {X 0,Y 266.675,Z 949.842,A -85,B 0,C 180,E1 12716.497,E2 12716.497} C_VEL
LIN {X 0,Y 262.569,Z 959.212,A -85,B 0,C 180,E1 12712.146,E2 12712.146} C_VEL
LIN {X 0,Y 259.623,Z 966.541,A -85,B 0,C 180,E1 12707.712,E2 12707.712} C_VEL
LIN {X 0,Y 257.719,Z 972.03,A -85,B 0,C 180,E1 12703.231,E2 12703.231} C_VEL
LIN {X 0,Y 256.69,Z 975.843,A -85,B 0,C 180,E1 12698.737,E2 12698.737} C_VEL
LIN {X 0,Y 256.271,Z 978.088,A -85,B 0,C 180,E1 12694.25,E2 12694.25} C_VEL
LIN {X 0,Y 256.195,Z 978.837,A -85,B 0,C 180,E1 12689.999,E2 12689.999} C_VEL
LIN {X 0,Y 256.266,Z 978.122,A -85,B 0,C 180,E1 12685.748,E2 12685.748} C_VEL
LIN {X 0,Y 256.679,Z 975.921,A -85,B 0,C 180,E1 12681.261,E2 12681.261} C_VEL
LIN {X 0,Y 257.695,Z 972.15,A -85,B 0,C 180,E1 12676.765,E2 12676.765} C_VEL
LIN {X 0,Y 259.58,Z 966.705,A -85,B 0,C 180,E1 12672.283,E2 12672.283} C_VEL
LIN {X 0,Y 262.642,Z 959.105,A -85,B 0,C 180,E1 12667.682,E2 12667.682} C_VEL
LIN {X 0,Y 266.596,Z 950.084,A -85,B 0,C 180,E1 12663.492,E2 12663.492} C_VEL
LIN {X 0,Y 271.304,Z 939.723,A -85,B 0,C 180,E1 12659.674,E2 12659.674} C_VEL
LIN {X 0,Y 276.646,Z 927.975,A -85,B 0,C 180,E1 12656.178,E2 12656.178} C_VEL
LIN {X 0,Y 282.852,Z 913.945,A -85,B 0,C 180,E1 12652.808,E2 12652.808} C_VEL
LIN {X 0,Y 289.012,Z 899.208,A -85,B 0,C 180,E1 12649.947,E2 12649.947} C_VEL
LIN {X 0,Y 294.97,Z 883.824,A -85,B 0,C 180,E1 12647.508,E2 12647.508} C_VEL
LIN {X 0,Y 300.876,Z 866.933,A -85,B 0,C 180,E1 12645.33,E2 12645.33} C_VEL
LIN {X 0,Y 306.434,Z 848.719,A -85,B 0,C 180,E1 12643.447,E2 12643.447} C_VEL
LIN {X 0,Y 311.249,Z 830.214,A -85,B 0,C 180,E1 12641.927,E2 12641.927} C_VEL
LIN {X 0,Y 315.269,Z 811.415,A -85,B 0,C 180,E1 12640.712,E2 12640.712} C_VEL
LIN {X 0,Y 318.692,Z 790.846,A -85,B 0,C 180,E1 12639.712,E2 12639.712} C_VEL
LIN {X 0,Y 321.035,Z 770.732,A -85,B 0,C 180,E1 12639.019,E2 12639.019} C_VEL
LIN {X 0,Y 322.146,Z 755.753,A -85,B 0,C 180,E1 12638.659,E2 12638.659} C_VEL
LIN {X 0,Y 321.992,Z 748.176,A -85,B 0,C 180,E1 12638.357,E2 12638.357} C_VEL
LIN {X 0,Y 319.421,Z 728.402,A -85,B 0,C 180,E1 12637.043,E2 12637.043} C_VEL
LIN {X 0,Y 319.391,Z 721.888,A -85,B 0,C 180,E1 12636.796,E2 12636.796} C_VEL
LIN {X 0,Y 323.906,Z 651.05,A -85,B 0,C 180,E1 12635.257,E2 12635.257} C_VEL
LIN {X 0,Y 317.545,Z 660.185,A -85,B 0,C 180,E1 12633.953,E2 12633.953} C_VEL
LIN {X 0,Y 316.67,Z 661.625,A -85,B 0,C 180,E1 12633.773,E2 12633.773} C_VEL
LIN {X 0,Y 310.535,Z 684.086,A -85,B 0,C 180,E1 12632.98,E2 12632.98} C_VEL
LIN {X 0,Y 306.022,Z 697.596,A -85,B 0,C 180,E1 12632.235,E2 12632.235} C_VEL
LIN {X 0,Y 302.436,Z 706.146,A -85,B 0,C 180,E1 12631.517,E2 12631.517} C_VEL
LIN {X 0,Y 296.254,Z 730.167,A -85,B 0,C 180,E1 12630.639,E2 12630.639} C_VEL
LIN {X 0,Y 291.283,Z 746.372,A -85,B 0,C 180,E1 12629.736,E2 12629.736} C_VEL
LIN {X 0,Y 287.95,Z 754.774,A -85,B 0,C 180,E1 12628.973,E2 12628.973} C_VEL
LIN {X 0,Y 286.546,Z 757.816,A -85,B 0,C 180,E1 12628.615,E2 12628.615} C_VEL
LIN {X 0,Y 281.909,Z 774.923,A -85,B 0,C 180,E1 12627.89,E2 12627.89} C_VEL
LIN {X 0,Y 278.179,Z 784.751,A -85,B 0,C 180,E1 12627.247,E2 12627.247} C_VEL
LIN {X 0,Y 274.925,Z 790.984,A -85,B 0,C 180,E1 12626.532,E2 12626.532} C_VEL
LIN {X 0,Y 272.372,Z 794.442,A -85,B 0,C 180,E1 12625.83,E2 12625.83} C_VEL
LIN {X 0,Y 268.745,Z 802.545,A -85,B 0,C 180,E1 12625.254,E2 12625.254} C_VEL
LIN {X 0,Y 265.273,Z 808.378,A -85,B 0,C 180,E1 12624.495,E2 12624.495} C_VEL
LIN {X 0,Y 263.462,Z 810.66,A -85,B 0,C 180,E1 12623.959,E2 12623.959} C_VEL
LIN {X 0,Y 262.078,Z 811.409,A -85,B 0,C 180,E1 12623.377,E2 12623.377} C_VEL
LIN {X 0,Y 261.88,Z 811.523,A -85,B 0,C 180,E1 12623.247,E2 12623.247} C_VEL
LIN {X 0,Y 260.08,Z 828.436,A -85,B 0,C 180,E1 12621.422,E2 12621.422} C_VEL
LIN {X 0,Y 258.11,Z 844.268,A -85,B 0,C 180,E1 12619.225,E2 12619.225} C_VEL
LIN {X 0,Y 256.218,Z 858.372,A -85,B 0,C 180,E1 12616.785,E2 12616.785} C_VEL
LIN {X 0,Y 254.498,Z 871.011,A -85,B 0,C 180,E1 12614.098,E2 12614.098} C_VEL
LIN {X 0,Y 252.954,Z 882.943,A -85,B 0,C 180,E1 12610.937,E2 12610.937} C_VEL
LIN {X 0,Y 251.884,Z 892.693,A -85,B 0,C 180,E1 12607.757,E2 12607.757} C_VEL
LIN {X 0,Y 251.209,Z 901.59,A -85,B 0,C 180,E1 12604.109,E2 12604.109} C_VEL
LIN {X 0,Y 251.078,Z 908.398,A -85,B 0,C 180,E1 12600.457,E2 12600.457} C_VEL
LIN {X 0,Y 251.484,Z 913.49,A -85,B 0,C 180,E1 12596.81,E2 12596.81} C_VEL
LIN {X 0,Y 252.627,Z 917.232,A -85,B 0,C 180,E1 12592.724,E2 12592.724} C_VEL
LIN {X 0,Y 254.48,Z 918.971,A -85,B 0,C 180,E1 12588.9,E2 12588.9} C_VEL
LIN {X 0,Y 257.212,Z 919.061,A -85,B 0,C 180,E1 12585.134,E2 12585.134} C_VEL
LIN {X 0,Y 261.345,Z 917.184,A -85,B 0,C 180,E1 12581.023,E2 12581.023} C_VEL
LIN {X 0,Y 266.689,Z 913.242,A -85,B 0,C 180,E1 12577.051,E2 12577.051} C_VEL
LIN {X 0,Y 272.909,Z 907.565,A -85,B 0,C 180,E1 12573.451,E2 12573.451} C_VEL
LIN {X 0,Y 280.249,Z 899.888,A -85,B 0,C 180,E1 12570.034,E2 12570.034} C_VEL
LIN {X 0,Y 288.237,Z 890.712,A -85,B 0,C 180,E1 12567.002,E2 12567.002} C_VEL
LIN {X 0,Y 297.318,Z 879.608,A -85,B 0,C 180,E1 12564.187,E2 12564.187} C_VEL
LIN {X 0,Y 307.582,Z 866.381,A -85,B 0,C 180,E1 12561.62,E2 12561.62} C_VEL
LIN {X 0,Y 313.573,Z 858.525,A -85,B 0,C 180,E1 12560.378,E2 12560.378} C_VEL
LIN {X 0,Y 302.286,Z 874.45,A -85,B 0,C 180,E1 12558.378,E2 12558.378} C_VEL
LIN {X 0,Y 292.147,Z 888.759,A -85,B 0,C 180,E1 12556.118,E2 12556.118} C_VEL
LIN {X 0,Y 285.648,Z 906.479,A -85,B 0,C 180,E1 12553.875,E2 12553.875} C_VEL
LIN {X 0,Y 278.968,Z 922.955,A -85,B 0,C 180,E1 12551.262,E2 12551.262} C_VEL
LIN {X 0,Y 272.555,Z 937.897,A -85,B 0,C 180,E1 12548.315,E2 12548.315} C_VEL
LIN {X 0,Y 266.504,Z 951.425,A -85,B 0,C 180,E1 12545.032,E2 12545.032} C_VEL
LIN {X 0,Y 260.79,Z 964.24,A -85,B 0,C 180,E1 12541.172,E2 12541.172} C_VEL
LIN {X 0,Y 256.131,Z 975.026,A -85,B 0,C 180,E1 12537.122,E2 12537.122} C_VEL
LIN {X 0,Y 252.539,Z 984.153,A -85,B 0,C 180,E1 12532.832,E2 12532.832} C_VEL
LIN {X 0,Y 250.02,Z 991.888,A -85,B 0,C 180,E1 12528.177,E2 12528.177} C_VEL
LIN {X 0,Y 248.607,Z 997.962,A -85,B 0,C 180,E1 12523.254,E2 12523.254} C_VEL
LIN {X 0,Y 248.203,Z 1001.735,A -85,B 0,C 180,E1 12518.807,E2 12518.807} C_VEL
LIN {X 0,Y 248.263,Z 1004.016,A -85,B 0,C 180,E1 12514.39,E2 12514.39} C_VEL
LIN {X 0,Y 248.369,Z 1004.786,A -85,B 0,C 180,E1 12510.463,E2 12510.463} C_VEL
LIN {X 0,Y 248.285,Z 1004.225,A -85,B 0,C 180,E1 12506.307,E2 12506.307} C_VEL
LIN {X 0,Y 248.177,Z 1002.379,A -85,B 0,C 180,E1 12502.128,E2 12502.128} C_VEL
LIN {X 0,Y 248.445,Z 998.833,A -85,B 0,C 180,E1 12497.686,E2 12497.686} C_VEL
LIN {X 0,Y 249.547,Z 993.433,A -85,B 0,C 180,E1 12492.994,E2 12492.994} C_VEL
LIN {X 0,Y 251.759,Z 986.196,A -85,B 0,C 180,E1 12488.326,E2 12488.326} C_VEL
LIN {X 0,Y 255.067,Z 977.485,A -85,B 0,C 180,E1 12483.959,E2 12483.959} C_VEL
LIN {X 0,Y 259.35,Z 967.402,A -85,B 0,C 180,E1 12479.923,E2 12479.923} C_VEL
LIN {X 0,Y 264.759,Z 955.198,A -85,B 0,C 180,E1 12476.02,E2 12476.02} C_VEL
LIN {X 0,Y 270.779,Z 941.692,A -85,B 0,C 180,E1 12472.55,E2 12472.55} C_VEL
LIN {X 0,Y 277.132,Z 927.03,A -85,B 0,C 180,E1 12469.504,E2 12469.504} C_VEL
LIN {X 0,Y 283.604,Z 911.251,A -85,B 0,C 180,E1 12466.848,E2 12466.848} C_VEL
LIN {X 0,Y 290.164,Z 893.898,A -85,B 0,C 180,E1 12464.498,E2 12464.498} C_VEL
LIN {X 0,Y 296.121,Z 876.397,A -85,B 0,C 180,E1 12462.603,E2 12462.603} C_VEL
LIN {X 0,Y 301.565,Z 858.181,A -85,B 0,C 180,E1 12461.032,E2 12461.032} C_VEL
LIN {X 0,Y 306.339,Z 839.233,A -85,B 0,C 180,E1 12459.771,E2 12459.771} C_VEL
LIN {X 0,Y 310.397,Z 819.339,A -85,B 0,C 180,E1 12458.774,E2 12458.774} C_VEL
LIN {X 0,Y 313.539,Z 798.389,A -85,B 0,C 180,E1 12458.022,E2 12458.022} C_VEL
LIN {X 0,Y 315.674,Z 775.271,A -85,B 0,C 180,E1 12457.476,E2 12457.476} C_VEL
LIN {X 0,Y 318.835,Z 746.478,A -85,B 0,C 180,E1 12457.173,E2 12457.173} C_VEL
LIN {X 0,Y 321.503,Z 726.625,A -85,B 0,C 180,E1 12457.081,E2 12457.081} C_VEL
LIN {X 0,Y 316.05,Z 707.314,A -85,B 0,C 180,E1 12455.029,E2 12455.029} C_VEL
LIN {X 0,Y 311.474,Z 686.895,A -85,B 0,C 180,E1 12452.991,E2 12452.991} C_VEL
LIN {X 0,Y 308.327,Z 666.945,A -85,B 0,C 180,E1 12451.228,E2 12451.228} C_VEL
LIN {X 0,Y 305.899,Z 646.529,A -85,B 0,C 180,E1 12449.547,E2 12449.547} C_VEL
LIN {X 0,Y 305.798,Z 641.954,A -85,B 0,C 180,E1 12449.193,E2 12449.193} C_VEL
LIN {X 0,Y 311.799,Z 613.707,A -85,B 0,C 180,E1 12445.856,E2 12445.856} C_VEL
LIN {X 0,Y 312.447,Z 610.653,A -85,B 0,C 180,E1 12445.493,E2 12445.493} C_VEL
LIN {X 0,Y 305.194,Z 594.011,A -85,B 0,C 180,E1 12441.526,E2 12441.526} C_VEL
LIN {X 0,Y 297.756,Z 577.462,A -85,B 0,C 180,E1 12437.187,E2 12437.187} C_VEL
LIN {X 0,Y 290.01,Z 560.928,A -85,B 0,C 180,E1 12432.342,E2 12432.342} C_VEL
LIN {X 0,Y 283.365,Z 547.384,A -85,B 0,C 180,E1 12427.909,E2 12427.909} C_VEL
LIN {X 0,Y 279.806,Z 539.948,A -85,B 0,C 180,E1 12425.228,E2 12425.228} C_VEL
LIN {X 0,Y 279.518,Z 533.723,A -85,B 0,C 180,E1 12422.05,E2 12422.05} C_VEL
LIN {X 0,Y 280.25,Z 526.921,A -85,B 0,C 180,E1 12418.057,E2 12418.057} C_VEL
LIN {X 0,Y 281.767,Z 522.643,A -85,B 0,C 180,E1 12414.655,E2 12414.655} C_VEL
LIN {X 0,Y 283.451,Z 523.866,A -85,B 0,C 180,E1 12411.48,E2 12411.48} C_VEL
LIN {X 0,Y 285.915,Z 527.821,A -85,B 0,C 180,E1 12408.093,E2 12408.093} C_VEL
LIN {X 0,Y 287.984,Z 529.791,A -85,B 0,C 180,E1 12406.036,E2 12406.036} C_VEL
LIN {X 0,Y 291.375,Z 534.287,A -85,B 0,C 180,E1 12403.144,E2 12403.144} C_VEL
LIN {X 0,Y 296.489,Z 541.114,A -85,B 0,C 180,E1 12399.623,E2 12399.623} C_VEL
LIN {X 0,Y 300.573,Z 546.722,A -85,B 0,C 180,E1 12397.25,E2 12397.25} C_VEL
LIN {X 0,Y 306.267,Z 554.754,A -85,B 0,C 180,E1 12394.369,E2 12394.369} C_VEL
LIN {X 0,Y 313.456,Z 565.719,A -85,B 0,C 180,E1 12391.206,E2 12391.206} C_VEL
LIN {X 0,Y 320.992,Z 578.341,A -85,B 0,C 180,E1 12388.288,E2 12388.288} C_VEL
LIN {X 0,Y 327.886,Z 590.944,A -85,B 0,C 180,E1 12385.882,E2 12385.882} C_VEL
LIN {X 0,Y 315.987,Z 770.492,A -85,B 0,C 180,E1 12382.015,E2 12382.015} C_VEL
LIN {X 0,Y 313.583,Z 790.796,A -85,B 0,C 180,E1 12381.321,E2 12381.321} C_VEL
LIN {X 0,Y 310.06,Z 811.453,A -85,B 0,C 180,E1 12380.32,E2 12380.32} C_VEL
LIN {X 0,Y 305.761,Z 830.905,A -85,B 0,C 180,E1 12379.057,E2 12379.057} C_VEL
LIN {X 0,Y 300.842,Z 849.186,A -85,B 0,C 180,E1 12377.545,E2 12377.545} C_VEL
LIN {X 0,Y 295.062,Z 867.469,A -85,B 0,C 180,E1 12375.642,E2 12375.642} C_VEL
LIN {X 0,Y 288.837,Z 884.632,A -85,B 0,C 180,E1 12373.403,E2 12373.403} C_VEL
LIN {X 0,Y 282.557,Z 900.193,A -85,B 0,C 180,E1 12370.891,E2 12370.891} C_VEL
LIN {X 0,Y 276.156,Z 914.835,A -85,B 0,C 180,E1 12367.987,E2 12367.987} C_VEL
LIN {X 0,Y 269.899,Z 928.359,A -85,B 0,C 180,E1 12364.672,E2 12364.672} C_VEL
LIN {X 0,Y 264.114,Z 940.461,A -85,B 0,C 180,E1 12360.986,E2 12360.986} C_VEL
LIN {X 0,Y 259.181,Z 950.759,A -85,B 0,C 180,E1 12357.077,E2 12357.077} C_VEL
LIN {X 0,Y 255.069,Z 959.629,A -85,B 0,C 180,E1 12352.834,E2 12352.834} C_VEL
LIN {X 0,Y 251.916,Z 966.959,A -85,B 0,C 180,E1 12348.272,E2 12348.272} C_VEL
LIN {X 0,Y 249.864,Z 972.446,A -85,B 0,C 180,E1 12343.655,E2 12343.655} C_VEL
LIN {X 0,Y 248.75,Z 976.257,A -85,B 0,C 180,E1 12339.018,E2 12339.018} C_VEL
LIN {X 0,Y 248.29,Z 978.5,A -85,B 0,C 180,E1 12334.387,E2 12334.387} C_VEL
LIN {X 0,Y 248.205,Z 979.249,A -85,B 0,C 180,E1 12329.999,E2 12329.999} C_VEL
LIN {X 0,Y 248.286,Z 978.533,A -85,B 0,C 180,E1 12325.611,E2 12325.611} C_VEL
LIN {X 0,Y 248.738,Z 976.334,A -85,B 0,C 180,E1 12320.979,E2 12320.979} C_VEL
LIN {X 0,Y 249.839,Z 972.565,A -85,B 0,C 180,E1 12316.341,E2 12316.341} C_VEL
LIN {X 0,Y 251.873,Z 967.12,A -85,B 0,C 180,E1 12311.722,E2 12311.722} C_VEL
LIN {X 0,Y 255.042,Z 959.744,A -85,B 0,C 180,E1 12307.116,E2 12307.116} C_VEL
LIN {X 0,Y 259.101,Z 950.998,A -85,B 0,C 180,E1 12302.911,E2 12302.911} C_VEL
LIN {X 0,Y 264.021,Z 940.753,A -85,B 0,C 180,E1 12298.999,E2 12298.999} C_VEL
LIN {X 0,Y 269.601,Z 929.112,A -85,B 0,C 180,E1 12295.419,E2 12295.419} C_VEL
LIN {X 0,Y 275.641,Z 916.16,A -85,B 0,C 180,E1 12292.19,E2 12292.19} C_VEL
LIN {X 0,Y 281.987,Z 901.781,A -85,B 0,C 180,E1 12289.274,E2 12289.274} C_VEL
LIN {X 0,Y 288.469,Z 885.854,A -85,B 0,C 180,E1 12286.662,E2 12286.662} C_VEL
LIN {X 0,Y 294.665,Z 868.847,A -85,B 0,C 180,E1 12284.415,E2 12284.415} C_VEL
LIN {X 0,Y 300.155,Z 851.748,A -85,B 0,C 180,E1 12282.591,E2 12282.591} C_VEL
LIN {X 0,Y 305.338,Z 833.006,A -85,B 0,C 180,E1 12280.991,E2 12280.991} C_VEL
LIN {X 0,Y 309.821,Z 813.217,A -85,B 0,C 180,E1 12279.672,E2 12279.672} C_VEL
LIN {X 0,Y 313.322,Z 793.445,A -85,B 0,C 180,E1 12278.68,E2 12278.68} C_VEL
LIN {X 0,Y 315.904,Z 772.934,A -85,B 0,C 180,E1 12277.944,E2 12277.944} C_VEL
LIN {X 0,Y 319.013,Z 727.804,A -85,B 0,C 180,E1 12276.923,E2 12276.923} C_VEL
LIN {X 0,Y 319.391,Z 721.888,A -85,B 0,C 180,E1 12276.796,E2 12276.796} C_VEL
LIN {X 0,Y 319.287,Z 714.313,A -85,B 0,C 180,E1 12276.489,E2 12276.489} C_VEL
LIN {X 0,Y 316.92,Z 694.562,A -85,B 0,C 180,E1 12275.141,E2 12275.141} C_VEL
LIN {X 0,Y 316.924,Z 688.05,A -85,B 0,C 180,E1 12274.889,E2 12274.889} C_VEL
LIN {X 0,Y 317.734,Z 675.253,A -85,B 0,C 180,E1 12274.6,E2 12274.6} C_VEL
LIN {X 0,Y 312.08,Z 694.029,A -85,B 0,C 180,E1 12273.826,E2 12273.826} C_VEL
LIN {X 0,Y 307.672,Z 705.606,A -85,B 0,C 180,E1 12273.063,E2 12273.063} C_VEL
LIN {X 0,Y 305.955,Z 709.653,A -85,B 0,C 180,E1 12272.735,E2 12272.735} C_VEL
LIN {X 0,Y 299.677,Z 733.478,A -85,B 0,C 180,E1 12271.884,E2 12271.884} C_VEL
LIN {X 0,Y 294.525,Z 749.85,A -85,B 0,C 180,E1 12270.995,E2 12270.995} C_VEL
LIN {X 0,Y 290.8,Z 759.072,A -85,B 0,C 180,E1 12270.189,E2 12270.189} C_VEL
LIN {X 0,Y 289.613,Z 761.801,A -85,B 0,C 180,E1 12269.914,E2 12269.914} C_VEL
LIN {X 0,Y 284.73,Z 778.5,A -85,B 0,C 180,E1 12269.231,E2 12269.231} C_VEL
LIN {X 0,Y 280.648,Z 788.638,A -85,B 0,C 180,E1 12268.589,E2 12268.589} C_VEL
LIN {X 0,Y 276.772,Z 795.656,A -85,B 0,C 180,E1 12267.835,E2 12267.835} C_VEL
LIN {X 0,Y 273.957,Z 799.776,A -85,B 0,C 180,E1 12267.163,E2 12267.163} C_VEL
LIN {X 0,Y 269.66,Z 808.218,A -85,B 0,C 180,E1 12266.509,E2 12266.509} C_VEL
LIN {X 0,Y 265.569,Z 814.335,A -85,B 0,C 180,E1 12265.657,E2 12265.657} C_VEL
LIN {X 0,Y 262.469,Z 817.671,A -85,B 0,C 180,E1 12264.774,E2 12264.774} C_VEL
LIN {X 0,Y 261.441,Z 818.738,A -85,B 0,C 180,E1 12264.462,E2 12264.462} C_VEL
LIN {X 0,Y 257.761,Z 824.372,A -85,B 0,C 180,E1 12263.728,E2 12263.728} C_VEL
LIN {X 0,Y 254.648,Z 828.003,A -85,B 0,C 180,E1 12262.875,E2 12262.875} C_VEL
LIN {X 0,Y 252.696,Z 829.342,A -85,B 0,C 180,E1 12262.08,E2 12262.08} C_VEL
LIN {X 0,Y 252.27,Z 829.532,A -85,B 0,C 180,E1 12261.792,E2 12261.792} C_VEL
LIN {X 0,Y 250.307,Z 844.905,A -85,B 0,C 180,E1 12259.606,E2 12259.606} C_VEL
LIN {X 0,Y 248.349,Z 859.045,A -85,B 0,C 180,E1 12257.092,E2 12257.092} C_VEL
LIN {X 0,Y 246.44,Z 872.668,A -85,B 0,C 180,E1 12254.09,E2 12254.09} C_VEL
LIN {X 0,Y 244.895,Z 884.564,A -85,B 0,C 180,E1 12250.825,E2 12250.825} C_VEL
LIN {X 0,Y 243.839,Z 894.282,A -85,B 0,C 180,E1 12247.54,E2 12247.54} C_VEL
LIN {X 0,Y 243.199,Z 903.119,A -85,B 0,C 180,E1 12243.772,E2 12243.772} C_VEL
LIN {X 0,Y 243.137,Z 909.935,A -85,B 0,C 180,E1 12240,E2 12240} C_VEL
LIN {X 0,Y 243.646,Z 915.041,A -85,B 0,C 180,E1 12236.236,E2 12236.236} C_VEL
LIN {X 0,Y 245.066,Z 918.996,A -85,B 0,C 180,E1 12231.791,E2 12231.791} C_VEL
LIN {X 0,Y 247.524,Z 920.801,A -85,B 0,C 180,E1 12227.401,E2 12227.401} C_VEL
LIN {X 0,Y 251.148,Z 920.534,A -85,B 0,C 180,E1 12223.105,E2 12223.105} C_VEL
LIN {X 0,Y 256.007,Z 918.273,A -85,B 0,C 180,E1 12218.942,E2 12218.942} C_VEL
LIN {X 0,Y 261.785,Z 914.269,A -85,B 0,C 180,E1 12215.157,E2 12215.157} C_VEL
LIN {X 0,Y 268.737,Z 908.443,A -85,B 0,C 180,E1 12211.561,E2 12211.561} C_VEL
LIN {X 0,Y 276.853,Z 900.721,A -85,B 0,C 180,E1 12208.178,E2 12208.178} C_VEL
LIN {X 0,Y 286.703,Z 890.397,A -85,B 0,C 180,E1 12204.871,E2 12204.871} C_VEL
LIN {X 0,Y 297.361,Z 878.577,A -85,B 0,C 180,E1 12202.025,E2 12202.025} C_VEL
LIN {X 0,Y 303.926,Z 871.003,A -85,B 0,C 180,E1 12200.538,E2 12200.538} C_VEL
LIN {X 0,Y 291.285,Z 886.93,A -85,B 0,C 180,E1 12198.15,E2 12198.15} C_VEL
LIN {X 0,Y 283.317,Z 897.153,A -85,B 0,C 180,E1 12196.235,E2 12196.235} C_VEL
LIN {X 0,Y 276.516,Z 914.056,A -85,B 0,C 180,E1 12193.826,E2 12193.826} C_VEL
LIN {X 0,Y 269.829,Z 929.399,A -85,B 0,C 180,E1 12191.102,E2 12191.102} C_VEL
LIN {X 0,Y 263.282,Z 943.67,A -85,B 0,C 180,E1 12187.97,E2 12187.97} C_VEL
LIN {X 0,Y 256.979,Z 956.994,A -85,B 0,C 180,E1 12184.346,E2 12184.346} C_VEL
LIN {X 0,Y 251.512,Z 968.684,A -85,B 0,C 180,E1 12180.384,E2 12180.384} C_VEL
LIN {X 0,Y 247.089,Z 978.647,A -85,B 0,C 180,E1 12176.174,E2 12176.174} C_VEL
LIN {X 0,Y 243.574,Z 987.47,A -85,B 0,C 180,E1 12171.43,E2 12171.43} C_VEL
LIN {X 0,Y 241.41,Z 994.293,A -85,B 0,C 180,E1 12166.607,E2 12166.607} C_VEL
LIN {X 0,Y 240.424,Z 999.082,A -85,B 0,C 180,E1 12162.003,E2 12162.003} C_VEL
LIN {X 0,Y 240.188,Z 1002.465,A -85,B 0,C 180,E1 12157.175,E2 12157.175} C_VEL
LIN {X 0,Y 240.321,Z 1004.104,A -85,B 0,C 180,E1 12152.863,E2 12152.863} C_VEL
LIN {X 0,Y 240.369,Z 1004.302,A -85,B 0,C 180,E1 12148.81,E2 12148.81} C_VEL
LIN {X 0,Y 240.23,Z 1003.377,A -85,B 0,C 180,E1 12144.748,E2 12144.748} C_VEL
LIN {X 0,Y 240.21,Z 1000.966,A -85,B 0,C 180,E1 12140.417,E2 12140.417} C_VEL
LIN {X 0,Y 240.801,Z 996.726,A -85,B 0,C 180,E1 12135.575,E2 12135.575} C_VEL
LIN {X 0,Y 242.426,Z 990.723,A -85,B 0,C 180,E1 12130.736,E2 12130.736} C_VEL
LIN {X 0,Y 245.329,Z 982.76,A -85,B 0,C 180,E1 12125.912,E2 12125.912} C_VEL
LIN {X 0,Y 249.561,Z 972.841,A -85,B 0,C 180,E1 12121.265,E2 12121.265} C_VEL
LIN {X 0,Y 254.964,Z 961.159,A -85,B 0,C 180,E1 12116.97,E2 12116.97} C_VEL
LIN {X 0,Y 261.103,Z 948.125,A -85,B 0,C 180,E1 12113.162,E2 12113.162} C_VEL
LIN {X 0,Y 267.388,Z 934.559,A -85,B 0,C 180,E1 12109.973,E2 12109.973} C_VEL
LIN {X 0,Y 274.235,Z 919.046,A -85,B 0,C 180,E1 12107.017,E2 12107.017} C_VEL
LIN {X 0,Y 281.313,Z 901.875,A -85,B 0,C 180,E1 12104.407,E2 12104.407} C_VEL
LIN {X 0,Y 287.84,Z 884.32,A -85,B 0,C 180,E1 12102.28,E2 12102.28} C_VEL
LIN {X 0,Y 293.726,Z 866.455,A -85,B 0,C 180,E1 12100.554,E2 12100.554} C_VEL
LIN {X 0,Y 299.055,Z 847.714,A -85,B 0,C 180,E1 12099.136,E2 12099.136} C_VEL
LIN {X 0,Y 303.73,Z 827.698,A -85,B 0,C 180,E1 12097.995,E2 12097.995} C_VEL
LIN {X 0,Y 307.361,Z 807.549,A -85,B 0,C 180,E1 12097.157,E2 12097.157} C_VEL
LIN {X 0,Y 309.858,Z 786.374,A -85,B 0,C 180,E1 12096.528,E2 12096.528} C_VEL
LIN {X 0,Y 312.38,Z 760.06,A -85,B 0,C 180,E1 12096.116,E2 12096.116} C_VEL
LIN {X 0,Y 316.38,Z 729.567,A -85,B 0,C 180,E1 12095.958,E2 12095.958} C_VEL
LIN {X 0,Y 316.203,Z 728.065,A -85,B 0,C 180,E1 12095.857,E2 12095.857} C_VEL
LIN {X 0,Y 310.598,Z 706.898,A -85,B 0,C 180,E1 12093.565,E2 12093.565} C_VEL
LIN {X 0,Y 306.248,Z 684.288,A -85,B 0,C 180,E1 12091.355,E2 12091.355} C_VEL
LIN {X 0,Y 303.154,Z 661.801,A -85,B 0,C 180,E1 12089.353,E2 12089.353} C_VEL
LIN {X 0,Y 300.987,Z 635.864,A -85,B 0,C 180,E1 12087.339,E2 12087.339} C_VEL
LIN {X 0,Y 301.094,Z 633.267,A -85,B 0,C 180,E1 12087.134,E2 12087.134} C_VEL
LIN {X 0,Y 305.621,Z 613.971,A -85,B 0,C 180,E1 12084.859,E2 12084.859} C_VEL
LIN {X 0,Y 298.094,Z 596.613,A -85,B 0,C 180,E1 12080.621,E2 12080.621} C_VEL
LIN {X 0,Y 290.684,Z 580.118,A -85,B 0,C 180,E1 12076.177,E2 12076.177} C_VEL
LIN {X 0,Y 283.535,Z 564.886,A -85,B 0,C 180,E1 12071.595,E2 12071.595} C_VEL
LIN {X 0,Y 280.122,Z 557.536,A -85,B 0,C 180,E1 12069.139,E2 12069.139} C_VEL
LIN {X 0,Y 278.687,Z 547.957,A -85,B 0,C 180,E1 12064.939,E2 12064.939} C_VEL
LIN {X 0,Y 278.523,Z 540.863,A -85,B 0,C 180,E1 12061.337,E2 12061.337} C_VEL
LIN {X 0,Y 279.406,Z 534.494,A -85,B 0,C 180,E1 12057.539,E2 12057.539} C_VEL
LIN {X 0,Y 280.856,Z 530.651,A -85,B 0,C 180,E1 12054.484,E2 12054.484} C_VEL
LIN {X 0,Y 282.34,Z 531.845,A -85,B 0,C 180,E1 12051.651,E2 12051.651} C_VEL
LIN {X 0,Y 284.946,Z 535.886,A -85,B 0,C 180,E1 12048.051,E2 12048.051} C_VEL
LIN {X 0,Y 286.687,Z 537.706,A -85,B 0,C 180,E1 12046.281,E2 12046.281} C_VEL
LIN {X 0,Y 290.757,Z 543.23,A -85,B 0,C 180,E1 12042.798,E2 12042.798} C_VEL
LIN {X 0,Y 294.689,Z 548.603,A -85,B 0,C 180,E1 12040.062,E2 12040.062} C_VEL
LIN {X 0,Y 298.678,Z 554.23,A -85,B 0,C 180,E1 12037.669,E2 12037.669} C_VEL
LIN {X 0,Y 304.074,Z 562.066,A -85,B 0,C 180,E1 12034.849,E2 12034.849} C_VEL
LIN {X 0,Y 311.02,Z 572.917,A -85,B 0,C 180,E1 12031.694,E2 12031.694} C_VEL
LIN {X 0,Y 318.843,Z 586.443,A -85,B 0,C 180,E1 12028.577,E2 12028.577} C_VEL
LIN {X 0,Y 323.212,Z 594.955,A -85,B 0,C 180,E1 12026.975,E2 12026.975} C_VEL
LIN {X 0,Y 311.122,Z 770.921,A -85,B 0,C 180,E1 12023.173,E2 12023.173} C_VEL
LIN {X 0,Y 308.63,Z 791.286,A -85,B 0,C 180,E1 12022.475,E2 12022.475} C_VEL
LIN {X 0,Y 305.002,Z 811.883,A -85,B 0,C 180,E1 12021.474,E2 12021.474} C_VEL
LIN {X 0,Y 300.571,Z 831.297,A -85,B 0,C 180,E1 12020.211,E2 12020.211} C_VEL
LIN {X 0,Y 295.483,Z 849.585,A -85,B 0,C 180,E1 12018.693,E2 12018.693} C_VEL
LIN {X 0,Y 289.495,Z 867.872,A -85,B 0,C 180,E1 12016.78,E2 12016.78} C_VEL
LIN {X 0,Y 283.033,Z 885.039,A -85,B 0,C 180,E1 12014.524,E2 12014.524} C_VEL
LIN {X 0,Y 276.501,Z 900.604,A -85,B 0,C 180,E1 12011.987,E2 12011.987} C_VEL
LIN {X 0,Y 269.822,Z 915.249,A -85,B 0,C 180,E1 12009.045,E2 12009.045} C_VEL
LIN {X 0,Y 263.115,Z 929.091,A -85,B 0,C 180,E1 12005.588,E2 12005.588} C_VEL
LIN {X 0,Y 256.869,Z 941.495,A -85,B 0,C 180,E1 12001.699,E2 12001.699} C_VEL
LIN {X 0,Y 251.618,Z 951.863,A -85,B 0,C 180,E1 11997.607,E2 11997.607} C_VEL
LIN {X 0,Y 247.406,Z 960.439,A -85,B 0,C 180,E1 11993.33,E2 11993.33} C_VEL
LIN {X 0,Y 244.099,Z 967.709,A -85,B 0,C 180,E1 11988.631,E2 11988.631} C_VEL
LIN {X 0,Y 241.866,Z 973.351,A -85,B 0,C 180,E1 11983.628,E2 11983.628} C_VEL
LIN {X 0,Y 240.733,Z 976.976,A -85,B 0,C 180,E1 11978.839,E2 11978.839} C_VEL
LIN {X 0,Y 240.283,Z 979.042,A -85,B 0,C 180,E1 11974.055,E2 11974.055} C_VEL
LIN {X 0,Y 240.207,Z 979.629,A -85,B 0,C 180,E1 11969.522,E2 11969.522} C_VEL
LIN {X 0,Y 240.32,Z 978.881,A -85,B 0,C 180,E1 11965.226,E2 11965.226} C_VEL
LIN {X 0,Y 240.845,Z 976.595,A -85,B 0,C 180,E1 11960.44,E2 11960.44} C_VEL
LIN {X 0,Y 242.162,Z 972.491,A -85,B 0,C 180,E1 11955.411,E2 11955.411} C_VEL
LIN {X 0,Y 244.464,Z 966.854,A -85,B 0,C 180,E1 11950.652,E2 11950.652} C_VEL
LIN {X 0,Y 247.742,Z 959.829,A -85,B 0,C 180,E1 11946.196,E2 11946.196} C_VEL
LIN {X 0,Y 252.422,Z 950.413,A -85,B 0,C 180,E1 11941.618,E2 11941.618} C_VEL
LIN {X 0,Y 258.066,Z 939.312,A -85,B 0,C 180,E1 11937.414,E2 11937.414} C_VEL
LIN {X 0,Y 264.086,Z 927.294,A -85,B 0,C 180,E1 11933.797,E2 11933.797} C_VEL
LIN {X 0,Y 270.554,Z 913.856,A -85,B 0,C 180,E1 11930.531,E2 11930.531} C_VEL
LIN {X 0,Y 277.31,Z 898.929,A -85,B 0,C 180,E1 11927.603,E2 11927.603} C_VEL
LIN {X 0,Y 284.147,Z 882.364,A -85,B 0,C 180,E1 11924.984,E2 11924.984} C_VEL
LIN {X 0,Y 290.421,Z 865.429,A -85,B 0,C 180,E1 11922.833,E2 11922.833} C_VEL
LIN {X 0,Y 296.183,Z 847.661,A -85,B 0,C 180,E1 11921.017,E2 11921.017} C_VEL
LIN {X 0,Y 301.393,Z 828.622,A -85,B 0,C 180,E1 11919.479,E2 11919.479} C_VEL
LIN {X 0,Y 305.656,Z 809.264,A -85,B 0,C 180,E1 11918.27,E2 11918.27} C_VEL
LIN {X 0,Y 309.04,Z 789.263,A -85,B 0,C 180,E1 11917.334,E2 11917.334} C_VEL
LIN {X 0,Y 311.48,Z 768.167,A -85,B 0,C 180,E1 11916.647,E2 11916.647} C_VEL
LIN {X 0,Y 316.924,Z 688.05,A -85,B 0,C 180,E1 11914.889,E2 11914.889} C_VEL
LIN {X 0,Y 316.114,Z 689.209,A -85,B 0,C 180,E1 11914.722,E2 11914.722} C_VEL
LIN {X 0,Y 314.085,Z 696.637,A -85,B 0,C 180,E1 11914.477,E2 11914.477} C_VEL
LIN {X 0,Y 310.908,Z 714.612,A -85,B 0,C 180,E1 11914.341,E2 11914.341} C_VEL
LIN {X 0,Y 310.042,Z 722.832,A -85,B 0,C 180,E1 11914.438,E2 11914.438} C_VEL
LIN {X 0,Y 306.345,Z 773.306,A -85,B 0,C 180,E1 11915.578,E2 11915.578} C_VEL
LIN {X 0,Y 303.668,Z 793.533,A -85,B 0,C 180,E1 11916.298,E2 11916.298} C_VEL
LIN {X 0,Y 300.004,Z 813.225,A -85,B 0,C 180,E1 11917.276,E2 11917.276} C_VEL
LIN {X 0,Y 295.366,Z 832.659,A -85,B 0,C 180,E1 11918.557,E2 11918.557} C_VEL
LIN {X 0,Y 290.105,Z 850.762,A -85,B 0,C 180,E1 11920.08,E2 11920.08} C_VEL
LIN {X 0,Y 283.911,Z 868.917,A -85,B 0,C 180,E1 11922.003,E2 11922.003} C_VEL
LIN {X 0,Y 277.264,Z 885.899,A -85,B 0,C 180,E1 11924.259,E2 11924.259} C_VEL
LIN {X 0,Y 270.427,Z 901.503,A -85,B 0,C 180,E1 11926.841,E2 11926.841} C_VEL
LIN {X 0,Y 263.467,Z 916.072,A -85,B 0,C 180,E1 11929.821,E2 11929.821} C_VEL
LIN {X 0,Y 256.792,Z 929.206,A -85,B 0,C 180,E1 11933.156,E2 11933.156} C_VEL
LIN {X 0,Y 250.359,Z 941.354,A -85,B 0,C 180,E1 11937.001,E2 11937.001} C_VEL
LIN {X 0,Y 245.021,Z 951.328,A -85,B 0,C 180,E1 11940.946,E2 11940.946} C_VEL
LIN {X 0,Y 240.334,Z 960.244,A -85,B 0,C 180,E1 11945.414,E2 11945.414} C_VEL
LIN {X 0,Y 236.678,Z 967.61,A -85,B 0,C 180,E1 11950.246,E2 11950.246} C_VEL
LIN {X 0,Y 234.256,Z 973.15,A -85,B 0,C 180,E1 11955.16,E2 11955.16} C_VEL
LIN {X 0,Y 232.918,Z 977.008,A -85,B 0,C 180,E1 11960.111,E2 11960.111} C_VEL
LIN {X 0,Y 232.341,Z 979.293,A -85,B 0,C 180,E1 11965.061,E2 11965.061} C_VEL
LIN {X 0,Y 232.217,Z 980.04,A -85,B 0,C 180,E1 11969.505,E2 11969.505} C_VEL
LIN {X 0,Y 232.302,Z 979.454,A -85,B 0,C 180,E1 11974.195,E2 11974.195} C_VEL
LIN {X 0,Y 232.796,Z 977.39,A -85,B 0,C 180,E1 11979.143,E2 11979.143} C_VEL
LIN {X 0,Y 234.029,Z 973.752,A -85,B 0,C 180,E1 11984.109,E2 11984.109} C_VEL
LIN {X 0,Y 236.432,Z 968.126,A -85,B 0,C 180,E1 11989.259,E2 11989.259} C_VEL
LIN {X 0,Y 240.054,Z 960.703,A -85,B 0,C 180,E1 11994.193,E2 11994.193} C_VEL
LIN {X 0,Y 244.826,Z 951.594,A -85,B 0,C 180,E1 11998.809,E2 11998.809} C_VEL
LIN {X 0,Y 250.331,Z 941.295,A -85,B 0,C 180,E1 12002.901,E2 12002.901} C_VEL
LIN {X 0,Y 256.508,Z 929.616,A -85,B 0,C 180,E1 12006.61,E2 12006.61} C_VEL
LIN {X 0,Y 263.146,Z 916.566,A -85,B 0,C 180,E1 12009.95,E2 12009.95} C_VEL
LIN {X 0,Y 270.071,Z 902.1,A -85,B 0,C 180,E1 12012.937,E2 12012.937} C_VEL
LIN {X 0,Y 277.087,Z 886.099,A -85,B 0,C 180,E1 12015.599,E2 12015.599} C_VEL
LIN {X 0,Y 283.77,Z 869.001,A -85,B 0,C 180,E1 12017.874,E2 12017.874} C_VEL
LIN {X 0,Y 289.667,Z 851.745,A -85,B 0,C 180,E1 12019.713,E2 12019.713} C_VEL
LIN {X 0,Y 294.911,Z 833.895,A -85,B 0,C 180,E1 12021.239,E2 12021.239} C_VEL
LIN {X 0,Y 299.689,Z 814.138,A -85,B 0,C 180,E1 12022.563,E2 12022.563} C_VEL
LIN {X 0,Y 303.394,Z 794.536,A -85,B 0,C 180,E1 12023.554,E2 12023.554} C_VEL
LIN {X 0,Y 306.158,Z 773.967,A -85,B 0,C 180,E1 12024.297,E2 12024.297} C_VEL
LIN {X 0,Y 309.353,Z 730.917,A -85,B 0,C 180,E1 12025.28,E2 12025.28} C_VEL
LIN {X 0,Y 318.6,Z 598.335,A -85,B 0,C 180,E1 12028.144,E2 12028.144} C_VEL
LIN {X 0,Y 311.282,Z 584.807,A -85,B 0,C 180,E1 12031.038,E2 12031.038} C_VEL
LIN {X 0,Y 304.7,Z 573.787,A -85,B 0,C 180,E1 12033.966,E2 12033.966} C_VEL
LIN {X 0,Y 298.261,Z 563.745,A -85,B 0,C 180,E1 12037.272,E2 12037.272} C_VEL
LIN {X 0,Y 294.273,Z 558.106,A -85,B 0,C 180,E1 12039.618,E2 12039.618} C_VEL
LIN {X 0,Y 291.459,Z 554.039,A -85,B 0,C 180,E1 12041.498,E2 12041.498} C_VEL
LIN {X 0,Y 288.076,Z 549.307,A -85,B 0,C 180,E1 12044.086,E2 12044.086} C_VEL
LIN {X 0,Y 284.733,Z 544.645,A -85,B 0,C 180,E1 12047.218,E2 12047.218} C_VEL
LIN {X 0,Y 281.567,Z 540.594,A -85,B 0,C 180,E1 12051.217,E2 12051.217} C_VEL
LIN {X 0,Y 280.899,Z 539.279,A -85,B 0,C 180,E1 12052.432,E2 12052.432} C_VEL
LIN {X 0,Y 279.862,Z 538.78,A -85,B 0,C 180,E1 12054.464,E2 12054.464} C_VEL
LIN {X 0,Y 278.271,Z 543.31,A -85,B 0,C 180,E1 12057.838,E2 12057.838} C_VEL
LIN {X 0,Y 277.498,Z 548.859,A -85,B 0,C 180,E1 12060.98,E2 12060.98} C_VEL
LIN {X 0,Y 277.545,Z 556.036,A -85,B 0,C 180,E1 12064.597,E2 12064.597} C_VEL
LIN {X 0,Y 279.033,Z 566.527,A -85,B 0,C 180,E1 12069.175,E2 12069.175} C_VEL
LIN {X 0,Y 283.575,Z 582.746,A -85,B 0,C 180,E1 12075.124,E2 12075.124} C_VEL
LIN {X 0,Y 290.333,Z 597.729,A -85,B 0,C 180,E1 12079.305,E2 12079.305} C_VEL
LIN {X 0,Y 298.289,Z 616.086,A -85,B 0,C 180,E1 12083.928,E2 12083.928} C_VEL
LIN {X 0,Y 298.704,Z 617.683,A -85,B 0,C 180,E1 12084.26,E2 12084.26} C_VEL
LIN {X 0,Y 296.743,Z 625.987,A -85,B 0,C 180,E1 12085.188,E2 12085.188} C_VEL
LIN {X 0,Y 297.782,Z 646.851,A -85,B 0,C 180,E1 12086.712,E2 12086.712} C_VEL
LIN {X 0,Y 299.933,Z 671.071,A -85,B 0,C 180,E1 12088.703,E2 12088.703} C_VEL
LIN {X 0,Y 303.36,Z 695.395,A -85,B 0,C 180,E1 12090.957,E2 12090.957} C_VEL
LIN {X 0,Y 308.302,Z 719.174,A -85,B 0,C 180,E1 12093.43,E2 12093.43} C_VEL
LIN {X 0,Y 311.436,Z 731.297,A -85,B 0,C 180,E1 12094.765,E2 12094.765} C_VEL
LIN {X 0,Y 307.282,Z 763.852,A -85,B 0,C 180,E1 12094.955,E2 12094.955} C_VEL
LIN {X 0,Y 304.918,Z 788.585,A -85,B 0,C 180,E1 12095.379,E2 12095.379} C_VEL
LIN {X 0,Y 302.182,Z 809.628,A -85,B 0,C 180,E1 12096.034,E2 12096.034} C_VEL
LIN {X 0,Y 298.076,Z 830.689,A -85,B 0,C 180,E1 12096.95,E2 12096.95} C_VEL
LIN {X 0,Y 293.099,Z 850.586,A -85,B 0,C 180,E1 12098.144,E2 12098.144} C_VEL
LIN {X 0,Y 287.489,Z 869.287,A -85,B 0,C 180,E1 12099.616,E2 12099.616} C_VEL
LIN {X 0,Y 281.002,Z 887.92,A -85,B 0,C 180,E1 12101.498,E2 12101.498} C_VEL
LIN {X 0,Y 274.051,Z 905.489,A -85,B 0,C 180,E1 12103.749,E2 12103.749} C_VEL
LIN {X 0,Y 266.818,Z 921.986,A -85,B 0,C 180,E1 12106.41,E2 12106.41} C_VEL
LIN {X 0,Y 259.814,Z 936.948,A -85,B 0,C 180,E1 12109.432,E2 12109.432} C_VEL
LIN {X 0,Y 253.151,Z 950.495,A -85,B 0,C 180,E1 12112.823,E2 12112.823} C_VEL
LIN {X 0,Y 246.777,Z 963.324,A -85,B 0,C 180,E1 12116.842,E2 12116.842} C_VEL
LIN {X 0,Y 241.578,Z 974.006,A -85,B 0,C 180,E1 12121.038,E2 12121.038} C_VEL
LIN {X 0,Y 237.427,Z 983.267,A -85,B 0,C 180,E1 12125.627,E2 12125.627} C_VEL
LIN {X 0,Y 234.455,Z 991.016,A -85,B 0,C 180,E1 12130.572,E2 12130.572} C_VEL
LIN {X 0,Y 232.789,Z 996.833,A -85,B 0,C 180,E1 12135.576,E2 12135.576} C_VEL
LIN {X 0,Y 232.214,Z 1000.765,A -85,B 0,C 180,E1 12140.406,E2 12140.406} C_VEL
LIN {X 0,Y 232.25,Z 1003.109,A -85,B 0,C 180,E1 12145.062,E2 12145.062} C_VEL
LIN {X 0,Y 232.383,Z 1003.914,A -85,B 0,C 180,E1 12149.015,E2 12149.015} C_VEL
LIN {X 0,Y 232.319,Z 1003.621,A -85,B 0,C 180,E1 12153.209,E2 12153.209} C_VEL
LIN {X 0,Y 232.195,Z 1002.05,A -85,B 0,C 180,E1 12157.424,E2 12157.424} C_VEL
LIN {X 0,Y 232.475,Z 998.665,A -85,B 0,C 180,E1 12162.42,E2 12162.42} C_VEL
LIN {X 0,Y 233.665,Z 993.559,A -85,B 0,C 180,E1 12167.431,E2 12167.431} C_VEL
LIN {X 0,Y 235.935,Z 987.049,A -85,B 0,C 180,E1 12172.16,E2 12172.16} C_VEL
LIN {X 0,Y 239.717,Z 978.226,A -85,B 0,C 180,E1 12177.043,E2 12177.043} C_VEL
LIN {X 0,Y 244.368,Z 968.396,A -85,B 0,C 180,E1 12181.309,E2 12181.309} C_VEL
LIN {X 0,Y 250.18,Z 956.661,A -85,B 0,C 180,E1 12185.384,E2 12185.384} C_VEL
LIN {X 0,Y 256.85,Z 943.255,A -85,B 0,C 180,E1 12189.098,E2 12189.098} C_VEL
LIN {X 0,Y 263.986,Z 928.378,A -85,B 0,C 180,E1 12192.392,E2 12192.392} C_VEL
LIN {X 0,Y 270.94,Z 913.038,A -85,B 0,C 180,E1 12195.118,E2 12195.118} C_VEL
LIN {X 0,Y 274.672,Z 904.48,A -85,B 0,C 180,E1 12196.42,E2 12196.42} C_VEL
LIN {X 0,Y 286.487,Z 890.814,A -85,B 0,C 180,E1 12199.232,E2 12199.232} C_VEL
LIN {X 0,Y 294.309,Z 881.965,A -85,B 0,C 180,E1 12200.747,E2 12200.747} C_VEL
LIN {X 0,Y 282.856,Z 893.352,A -85,B 0,C 180,E1 12203.569,E2 12203.569} C_VEL
LIN {X 0,Y 272.339,Z 903.181,A -85,B 0,C 180,E1 12206.837,E2 12206.837} C_VEL
LIN {X 0,Y 263.628,Z 910.6,A -85,B 0,C 180,E1 12210.209,E2 12210.209} C_VEL
LIN {X 0,Y 255.732,Z 916.494,A -85,B 0,C 180,E1 12214.031,E2 12214.031} C_VEL
LIN {X 0,Y 249.489,Z 920.262,A -85,B 0,C 180,E1 12217.87,E2 12217.87} C_VEL
LIN {X 0,Y 244.2,Z 922.345,A -85,B 0,C 180,E1 12222.117,E2 12222.117} C_VEL
LIN {X 0,Y 240.202,Z 922.481,A -85,B 0,C 180,E1 12226.521,E2 12226.521} C_VEL
LIN {X 0,Y 237.455,Z 920.589,A -85,B 0,C 180,E1 12231.037,E2 12231.037} C_VEL
LIN {X 0,Y 235.827,Z 916.574,A -85,B 0,C 180,E1 12235.624,E2 12235.624} C_VEL
LIN {X 0,Y 235.172,Z 910.696,A -85,B 0,C 180,E1 12240,E2 12240} C_VEL
LIN {X 0,Y 235.232,Z 903.609,A -85,B 0,C 180,E1 12243.9,E2 12243.9} C_VEL
LIN {X 0,Y 235.847,Z 895.156,A -85,B 0,C 180,E1 12247.552,E2 12247.552} C_VEL
LIN {X 0,Y 237.019,Z 884.576,A -85,B 0,C 180,E1 12251.19,E2 12251.19} C_VEL
LIN {X 0,Y 238.512,Z 873.349,A -85,B 0,C 180,E1 12254.32,E2 12254.32} C_VEL
LIN {X 0,Y 240.482,Z 859.604,A -85,B 0,C 180,E1 12257.419,E2 12257.419} C_VEL
LIN {X 0,Y 242.665,Z 844.475,A -85,B 0,C 180,E1 12260.187,E2 12260.187} C_VEL
LIN {X 0,Y 243.871,Z 844.18,A -85,B 0,C 180,E1 12260.898,E2 12260.898} C_VEL
LIN {X 0,Y 246.635,Z 841.757,A -85,B 0,C 180,E1 12261.899,E2 12261.899} C_VEL
LIN {X 0,Y 250.195,Z 837.53,A -85,B 0,C 180,E1 12262.808,E2 12262.808} C_VEL
LIN {X 0,Y 251.305,Z 836.189,A -85,B 0,C 180,E1 12263.073,E2 12263.073} C_VEL
LIN {X 0,Y 254.384,Z 833.801,A -85,B 0,C 180,E1 12264.128,E2 12264.128} C_VEL
LIN {X 0,Y 258.474,Z 829.135,A -85,B 0,C 180,E1 12265.149,E2 12265.149} C_VEL
LIN {X 0,Y 262.342,Z 823.867,A -85,B 0,C 180,E1 12265.91,E2 12265.91} C_VEL
LIN {X 0,Y 265.885,Z 820.228,A -85,B 0,C 180,E1 12266.825,E2 12266.825} C_VEL
LIN {X 0,Y 270.513,Z 813.836,A -85,B 0,C 180,E1 12267.757,E2 12267.757} C_VEL
LIN {X 0,Y 275.475,Z 804.999,A -85,B 0,C 180,E1 12268.489,E2 12268.489} C_VEL
LIN {X 0,Y 276.562,Z 803.209,A -85,B 0,C 180,E1 12268.681,E2 12268.681} C_VEL
LIN {X 0,Y 280.985,Z 796.586,A -85,B 0,C 180,E1 12269.557,E2 12269.557} C_VEL
LIN {X 0,Y 285.841,Z 786.751,A -85,B 0,C 180,E1 12270.307,E2 12270.307} C_VEL
LIN {X 0,Y 291.151,Z 771.537,A -85,B 0,C 180,E1 12270.992,E2 12270.992} C_VEL
LIN {X 0,Y 293.358,Z 764.199,A -85,B 0,C 180,E1 12271.289,E2 12271.289} C_VEL
LIN {X 0,Y 297.385,Z 754.743,A -85,B 0,C 180,E1 12272.128,E2 12272.128} C_VEL
LIN {X 0,Y 302.511,Z 739.238,A -85,B 0,C 180,E1 12272.993,E2 12272.993} C_VEL
LIN {X 0,Y 308.875,Z 716.079,A -85,B 0,C 180,E1 12273.841,E2 12273.841} C_VEL
LIN {X 0,Y 310.148,Z 711.599,A -85,B 0,C 180,E1 12274.01,E2 12274.01} C_VEL
LIN {X 0,Y 310.914,Z 710.128,A -85,B 0,C 180,E1 12274.161,E2 12274.161} C_VEL
LIN {X 0,Y 310.042,Z 722.832,A -85,B 0,C 180,E1 12274.438,E2 12274.438} C_VEL
LIN {X 0,Y 308.924,Z 731.629,A -85,B 0,C 180,E1 12274.488,E2 12274.488} C_VEL
LIN {X 0,Y 306.652,Z 741.466,A -85,B 0,C 180,E1 12274.262,E2 12274.262} C_VEL
LIN {X 0,Y 302.788,Z 753.314,A -85,B 0,C 180,E1 12273.668,E2 12273.668} C_VEL
LIN {X 0,Y 299.689,Z 761.271,A -85,B 0,C 180,E1 12273.113,E2 12273.113} C_VEL
LIN {X 0,Y 296.163,Z 769.203,A -85,B 0,C 180,E1 12272.459,E2 12272.459} C_VEL
LIN {X 0,Y 291.074,Z 784.6,A -85,B 0,C 180,E1 12271.893,E2 12271.893} C_VEL
LIN {X 0,Y 286.118,Z 795.689,A -85,B 0,C 180,E1 12271.276,E2 12271.276} C_VEL
LIN {X 0,Y 281.056,Z 804.254,A -85,B 0,C 180,E1 12270.49,E2 12270.49} C_VEL
LIN {X 0,Y 277.93,Z 808.557,A -85,B 0,C 180,E1 12269.886,E2 12269.886} C_VEL
LIN {X 0,Y 272.234,Z 818.146,A -85,B 0,C 180,E1 12269.133,E2 12269.133} C_VEL
LIN {X 0,Y 266.857,Z 825.172,A -85,B 0,C 180,E1 12268.171,E2 12268.171} C_VEL
LIN {X 0,Y 261.861,Z 830.485,A -85,B 0,C 180,E1 12267.025,E2 12267.025} C_VEL
LIN {X 0,Y 256.901,Z 836.576,A -85,B 0,C 180,E1 12266.091,E2 12266.091} C_VEL
LIN {X 0,Y 252.665,Z 840.755,A -85,B 0,C 180,E1 12265.01,E2 12265.01} C_VEL
LIN {X 0,Y 250.055,Z 842.869,A -85,B 0,C 180,E1 12264.183,E2 12264.183} C_VEL
LIN {X 0,Y 245.876,Z 847.382,A -85,B 0,C 180,E1 12263.212,E2 12263.212} C_VEL
LIN {X 0,Y 242.296,Z 850.462,A -85,B 0,C 180,E1 12262.057,E2 12262.057} C_VEL
LIN {X 0,Y 240.185,Z 851.831,A -85,B 0,C 180,E1 12261.171,E2 12261.171} C_VEL
LIN {X 0,Y 236.387,Z 855.685,A -85,B 0,C 180,E1 12260.036,E2 12260.036} C_VEL
LIN {X 0,Y 233.92,Z 857.432,A -85,B 0,C 180,E1 12258.957,E2 12258.957} C_VEL
LIN {X 0,Y 232.978,Z 857.674,A -85,B 0,C 180,E1 12258.258,E2 12258.258} C_VEL
LIN {X 0,Y 231.012,Z 870.984,A -85,B 0,C 180,E1 12255.309,E2 12255.309} C_VEL
LIN {X 0,Y 229.251,Z 883.648,A -85,B 0,C 180,E1 12251.829,E2 12251.829} C_VEL
LIN {X 0,Y 228.037,Z 894.008,A -85,B 0,C 180,E1 12248.32,E2 12248.32} C_VEL
LIN {X 0,Y 227.318,Z 903.008,A -85,B 0,C 180,E1 12244.541,E2 12244.541} C_VEL
LIN {X 0,Y 227.185,Z 910.965,A -85,B 0,C 180,E1 12240.253,E2 12240.253} C_VEL
LIN {X 0,Y 227.723,Z 916.636,A -85,B 0,C 180,E1 12236.224,E2 12236.224} C_VEL
LIN {X 0,Y 229.179,Z 921.116,A -85,B 0,C 180,E1 12231.723,E2 12231.723} C_VEL
LIN {X 0,Y 231.847,Z 923.771,A -85,B 0,C 180,E1 12227.041,E2 12227.041} C_VEL
LIN {X 0,Y 235.808,Z 924.395,A -85,B 0,C 180,E1 12222.48,E2 12222.48} C_VEL
LIN {X 0,Y 241.121,Z 923.106,A -85,B 0,C 180,E1 12218.087,E2 12218.087} C_VEL
LIN {X 0,Y 247.818,Z 919.93,A -85,B 0,C 180,E1 12213.911,E2 12213.911} C_VEL
LIN {X 0,Y 255.901,Z 914.884,A -85,B 0,C 180,E1 12209.992,E2 12209.992} C_VEL
LIN {X 0,Y 265.351,Z 907.964,A -85,B 0,C 180,E1 12206.365,E2 12206.365} C_VEL
LIN {X 0,Y 276.758,Z 898.586,A -85,B 0,C 180,E1 12202.892,E2 12202.892} C_VEL
LIN {X 0,Y 284.735,Z 891.655,A -85,B 0,C 180,E1 12200.902,E2 12200.902} C_VEL
LIN {X 0,Y 271.462,Z 905.337,A -85,B 0,C 180,E1 12198.076,E2 12198.076} C_VEL
LIN {X 0,Y 265.785,Z 911.45,A -85,B 0,C 180,E1 12196.558,E2 12196.558} C_VEL
LIN {X 0,Y 258.236,Z 927.455,A -85,B 0,C 180,E1 12193.721,E2 12193.721} C_VEL
LIN {X 0,Y 250.757,Z 942.39,A -85,B 0,C 180,E1 12190.396,E2 12190.396} C_VEL
LIN {X 0,Y 243.934,Z 955.446,A -85,B 0,C 180,E1 12186.76,E2 12186.76} C_VEL
LIN {X 0,Y 237.995,Z 966.807,A -85,B 0,C 180,E1 12182.818,E2 12182.818} C_VEL
LIN {X 0,Y 232.642,Z 977.324,A -85,B 0,C 180,E1 12178.215,E2 12178.215} C_VEL
LIN {X 0,Y 228.498,Z 986.219,A -85,B 0,C 180,E1 12173.194,E2 12173.194} C_VEL
LIN {X 0,Y 225.861,Z 993.139,A -85,B 0,C 180,E1 12168.054,E2 12168.054} C_VEL
LIN {X 0,Y 224.531,Z 998.246,A -85,B 0,C 180,E1 12162.866,E2 12162.866} C_VEL
LIN {X 0,Y 224.205,Z 1001.636,A -85,B 0,C 180,E1 12157.69,E2 12157.69} C_VEL
LIN {X 0,Y 224.332,Z 1003.28,A -85,B 0,C 180,E1 12153.067,E2 12153.067} C_VEL
LIN {X 0,Y 224.388,Z 1003.479,A -85,B 0,C 180,E1 12148.725,E2 12148.725} C_VEL
LIN {X 0,Y 224.234,Z 1002.549,A -85,B 0,C 180,E1 12144.372,E2 12144.372} C_VEL
LIN {X 0,Y 224.27,Z 999.964,A -85,B 0,C 180,E1 12139.469,E2 12139.469} C_VEL
LIN {X 0,Y 225.085,Z 995.62,A -85,B 0,C 180,E1 12134.279,E2 12134.279} C_VEL
LIN {X 0,Y 227.106,Z 989.512,A -85,B 0,C 180,E1 12129.109,E2 12129.109} C_VEL
LIN {X 0,Y 230.355,Z 981.98,A -85,B 0,C 180,E1 12124.276,E2 12124.276} C_VEL
LIN {X 0,Y 235.235,Z 971.993,A -85,B 0,C 180,E1 12119.334,E2 12119.334} C_VEL
LIN {X 0,Y 241.306,Z 960.314,A -85,B 0,C 180,E1 12114.835,E2 12114.835} C_VEL
LIN {X 0,Y 247.893,Z 947.732,A -85,B 0,C 180,E1 12111.009,E2 12111.009} C_VEL
LIN {X 0,Y 255.032,Z 933.721,A -85,B 0,C 180,E1 12107.6,E2 12107.6} C_VEL
LIN {X 0,Y 262.248,Z 918.775,A -85,B 0,C 180,E1 12104.681,E2 12104.681} C_VEL
LIN {X 0,Y 269.873,Z 901.724,A -85,B 0,C 180,E1 12102.028,E2 12102.028} C_VEL
LIN {X 0,Y 276.873,Z 884.322,A -85,B 0,C 180,E1 12099.881,E2 12099.881} C_VEL
LIN {X 0,Y 283.338,Z 866.071,A -85,B 0,C 180,E1 12098.102,E2 12098.102} C_VEL
LIN {X 0,Y 289.145,Z 846.927,A -85,B 0,C 180,E1 12096.656,E2 12096.656} C_VEL
LIN {X 0,Y 293.997,Z 827.372,A -85,B 0,C 180,E1 12095.546,E2 12095.546} C_VEL
LIN {X 0,Y 297.889,Z 807.079,A -85,B 0,C 180,E1 12094.703,E2 12094.703} C_VEL
LIN {X 0,Y 300.57,Z 785.831,A -85,B 0,C 180,E1 12094.071,E2 12094.071} C_VEL
LIN {X 0,Y 303.305,Z 758.829,A -85,B 0,C 180,E1 12093.669,E2 12093.669} C_VEL
LIN {X 0,Y 306.557,Z 732.841,A -85,B 0,C 180,E1 12093.505,E2 12093.505} C_VEL
LIN {X 0,Y 301.258,Z 709.814,A -85,B 0,C 180,E1 12090.946,E2 12090.946} C_VEL
LIN {X 0,Y 297.251,Z 684.473,A -85,B 0,C 180,E1 12088.422,E2 12088.422} C_VEL
LIN {X 0,Y 294.608,Z 657.374,A -85,B 0,C 180,E1 12086.045,E2 12086.045} C_VEL
LIN {X 0,Y 293.279,Z 629.64,A -85,B 0,C 180,E1 12083.941,E2 12083.941} C_VEL
LIN {X 0,Y 292.919,Z 621.041,A -85,B 0,C 180,E1 12083.272,E2 12083.272} C_VEL
LIN {X 0,Y 285.173,Z 600.987,A -85,B 0,C 180,E1 12077.865,E2 12077.865} C_VEL
LIN {X 0,Y 280.783,Z 587.027,A -85,B 0,C 180,E1 12073.488,E2 12073.488} C_VEL
LIN {X 0,Y 277.217,Z 571.319,A -85,B 0,C 180,E1 12067.512,E2 12067.512} C_VEL
LIN {X 0,Y 276.344,Z 561.44,A -85,B 0,C 180,E1 12063.037,E2 12063.037} C_VEL
LIN {X 0,Y 276.756,Z 554.426,A -85,B 0,C 180,E1 12059.379,E2 12059.379} C_VEL
LIN {X 0,Y 277.789,Z 549.625,A -85,B 0,C 180,E1 12056.492,E2 12056.492} C_VEL
LIN {X 0,Y 279.041,Z 546.663,A -85,B 0,C 180,E1 12054.138,E2 12054.138} C_VEL
LIN {X 0,Y 280.028,Z 547.5,A -85,B 0,C 180,E1 12052.202,E2 12052.202} C_VEL
LIN {X 0,Y 282.649,Z 551.665,A -85,B 0,C 180,E1 12048.367,E2 12048.367} C_VEL
LIN {X 0,Y 283.933,Z 553.151,A -85,B 0,C 180,E1 12046.975,E2 12046.975} C_VEL
LIN {X 0,Y 287.554,Z 558.366,A -85,B 0,C 180,E1 12043.641,E2 12043.641} C_VEL
LIN {X 0,Y 291.211,Z 563.682,A -85,B 0,C 180,E1 12040.911,E2 12040.911} C_VEL
LIN {X 0,Y 295.017,Z 569.338,A -85,B 0,C 180,E1 12038.477,E2 12038.477} C_VEL
LIN {X 0,Y 301.246,Z 578.988,A -85,B 0,C 180,E1 12035.069,E2 12035.069} C_VEL
LIN {X 0,Y 308.042,Z 590.666,A -85,B 0,C 180,E1 12031.871,E2 12031.871} C_VEL
LIN {X 0,Y 314.265,Z 602.457,A -85,B 0,C 180,E1 12029.27,E2 12029.27} C_VEL
LIN {X 0,Y 301.781,Z 771.881,A -85,B 0,C 180,E1 12025.596,E2 12025.596} C_VEL
LIN {X 0,Y 299.134,Z 792.163,A -85,B 0,C 180,E1 12024.9,E2 12024.9} C_VEL
LIN {X 0,Y 295.279,Z 812.735,A -85,B 0,C 180,E1 12023.9,E2 12023.9} C_VEL
LIN {X 0,Y 290.574,Z 832.082,A -85,B 0,C 180,E1 12022.641,E2 12022.641} C_VEL
LIN {X 0,Y 285.142,Z 850.383,A -85,B 0,C 180,E1 12021.117,E2 12021.117} C_VEL
LIN {X 0,Y 278.727,Z 868.68,A -85,B 0,C 180,E1 12019.19,E2 12019.19} C_VEL
LIN {X 0,Y 271.771,Z 885.855,A -85,B 0,C 180,E1 12016.909,E2 12016.909} C_VEL
LIN {X 0,Y 264.565,Z 901.753,A -85,B 0,C 180,E1 12014.267,E2 12014.267} C_VEL
LIN {X 0,Y 257.453,Z 916.075,A -85,B 0,C 180,E1 12011.315,E2 12011.315} C_VEL
LIN {X 0,Y 250.456,Z 929.28,A -85,B 0,C 180,E1 12007.935,E2 12007.935} C_VEL
LIN {X 0,Y 243.911,Z 941.094,A -85,B 0,C 180,E1 12004.165,E2 12004.165} C_VEL
LIN {X 0,Y 238.036,Z 951.513,A -85,B 0,C 180,E1 11999.989,E2 11999.989} C_VEL
LIN {X 0,Y 232.809,Z 960.883,A -85,B 0,C 180,E1 11995.161,E2 11995.161} C_VEL
LIN {X 0,Y 228.893,Z 968.34,A -85,B 0,C 180,E1 11990.086,E2 11990.086} C_VEL
LIN {X 0,Y 226.291,Z 973.939,A -85,B 0,C 180,E1 11984.848,E2 11984.848} C_VEL
LIN {X 0,Y 224.911,Z 977.652,A -85,B 0,C 180,E1 11979.724,E2 11979.724} C_VEL
LIN {X 0,Y 224.337,Z 979.802,A -85,B 0,C 180,E1 11974.6,E2 11974.6} C_VEL
LIN {X 0,Y 224.236,Z 980.483,A -85,B 0,C 180,E1 11969.999,E2 11969.999} C_VEL
LIN {X 0,Y 224.347,Z 979.77,A -85,B 0,C 180,E1 11965.141,E2 11965.141} C_VEL
LIN {X 0,Y 224.947,Z 977.574,A -85,B 0,C 180,E1 11960.016,E2 11960.016} C_VEL
LIN {X 0,Y 226.355,Z 973.809,A -85,B 0,C 180,E1 11954.892,E2 11954.892} C_VEL
LIN {X 0,Y 228.906,Z 968.366,A -85,B 0,C 180,E1 11949.812,E2 11949.812} C_VEL
LIN {X 0,Y 232.743,Z 961.063,A -85,B 0,C 180,E1 11944.829,E2 11944.829} C_VEL
LIN {X 0,Y 237.655,Z 952.241,A -85,B 0,C 180,E1 11940.233,E2 11940.233} C_VEL
LIN {X 0,Y 243.459,Z 941.992,A -85,B 0,C 180,E1 11936.044,E2 11936.044} C_VEL
LIN {X 0,Y 249.939,Z 930.368,A -85,B 0,C 180,E1 11932.26,E2 11932.26} C_VEL
LIN {X 0,Y 256.876,Z 917.383,A -85,B 0,C 180,E1 11928.865,E2 11928.865} C_VEL
LIN {X 0,Y 264.092,Z 902.992,A -85,B 0,C 180,E1 11925.841,E2 11925.841} C_VEL
LIN {X 0,Y 271.376,Z 887.054,A -85,B 0,C 180,E1 11923.153,E2 11923.153} C_VEL
LIN {X 0,Y 278.333,Z 869.959,A -85,B 0,C 180,E1 11920.854,E2 11920.854} C_VEL
LIN {X 0,Y 284.672,Z 852.119,A -85,B 0,C 180,E1 11918.938,E2 11918.938} C_VEL
LIN {X 0,Y 290.131,Z 834.141,A -85,B 0,C 180,E1 11917.404,E2 11917.404} C_VEL
LIN {X 0,Y 295.068,Z 814.309,A -85,B 0,C 180,E1 11916.08,E2 11916.08} C_VEL
LIN {X 0,Y 298.889,Z 794.613,A -85,B 0,C 180,E1 11915.092,E2 11915.092} C_VEL
LIN {X 0,Y 301.706,Z 774.209,A -85,B 0,C 180,E1 11914.359,E2 11914.359} C_VEL
LIN {X 0,Y 303.551,Z 750.746,A -85,B 0,C 180,E1 11913.783,E2 11913.783} C_VEL
LIN {X 0,Y 299.689,Z 761.271,A -85,B 0,C 180,E1 11913.113,E2 11913.113} C_VEL
LIN {X 0,Y 298.473,Z 765.464,A -85,B 0,C 180,E1 11912.948,E2 11912.948} C_VEL
LIN {X 0,Y 297.513,Z 772.923,A -85,B 0,C 180,E1 11913.075,E2 11913.075} C_VEL
LIN {X 0,Y 296.522,Z 781.264,A -85,B 0,C 180,E1 11913.337,E2 11913.337} C_VEL
LIN {X 0,Y 295.51,Z 784.886,A -85,B 0,C 180,E1 11913.294,E2 11913.294} C_VEL
LIN {X 0,Y 289.953,Z 797.468,A -85,B 0,C 180,E1 11912.697,E2 11912.697} C_VEL
LIN {X 0,Y 284.246,Z 807.175,A -85,B 0,C 180,E1 11911.935,E2 11911.935} C_VEL
LIN {X 0,Y 279.803,Z 813.184,A -85,B 0,C 180,E1 11911.209,E2 11911.209} C_VEL
LIN {X 0,Y 273.78,Z 822.744,A -85,B 0,C 180,E1 11910.469,E2 11910.469} C_VEL
LIN {X 0,Y 267.945,Z 830.091,A -85,B 0,C 180,E1 11909.51,E2 11909.51} C_VEL
LIN {X 0,Y 262.257,Z 835.847,A -85,B 0,C 180,E1 11908.35,E2 11908.35} C_VEL
LIN {X 0,Y 256.59,Z 842.421,A -85,B 0,C 180,E1 11907.318,E2 11907.318} C_VEL
LIN {X 0,Y 251.689,Z 846.861,A -85,B 0,C 180,E1 11906.165,E2 11906.165} C_VEL
LIN {X 0,Y 249.099,Z 848.92,A -85,B 0,C 180,E1 11905.435,E2 11905.435} C_VEL
LIN {X 0,Y 243.889,Z 854.107,A -85,B 0,C 180,E1 11904.203,E2 11904.203} C_VEL
LIN {X 0,Y 239.627,Z 857.294,A -85,B 0,C 180,E1 11902.834,E2 11902.834} C_VEL
LIN {X 0,Y 238.597,Z 857.894,A -85,B 0,C 180,E1 11902.417,E2 11902.417} C_VEL
LIN {X 0,Y 233.954,Z 862.16,A -85,B 0,C 180,E1 11901.039,E2 11901.039} C_VEL
LIN {X 0,Y 230.957,Z 864.16,A -85,B 0,C 180,E1 11899.736,E2 11899.736} C_VEL
LIN {X 0,Y 230.1,Z 864.592,A -85,B 0,C 180,E1 11899.284,E2 11899.284} C_VEL
LIN {X 0,Y 226.445,Z 867.83,A -85,B 0,C 180,E1 11898.004,E2 11898.004} C_VEL
LIN {X 0,Y 224.246,Z 869.256,A -85,B 0,C 180,E1 11896.848,E2 11896.848} C_VEL
LIN {X 0,Y 223.37,Z 869.586,A -85,B 0,C 180,E1 11896.046,E2 11896.046} C_VEL
LIN {X 0,Y 221.621,Z 881.768,A -85,B 0,C 180,E1 11892.772,E2 11892.772} C_VEL
LIN {X 0,Y 220.184,Z 893.359,A -85,B 0,C 180,E1 11888.882,E2 11888.882} C_VEL
LIN {X 0,Y 219.379,Z 902.726,A -85,B 0,C 180,E1 11884.968,E2 11884.968} C_VEL
LIN {X 0,Y 219.189,Z 910.731,A -85,B 0,C 180,E1 11880.785,E2 11880.785} C_VEL
LIN {X 0,Y 219.779,Z 917.492,A -85,B 0,C 180,E1 11876.087,E2 11876.087} C_VEL
LIN {X 0,Y 221.327,Z 922.23,A -85,B 0,C 180,E1 11871.427,E2 11871.427} C_VEL
LIN {X 0,Y 223.809,Z 925.009,A -85,B 0,C 180,E1 11867.093,E2 11867.093} C_VEL
LIN {X 0,Y 227.873,Z 926.218,A -85,B 0,C 180,E1 11862.377,E2 11862.377} C_VEL
LIN {X 0,Y 233.351,Z 925.527,A -85,B 0,C 180,E1 11857.849,E2 11857.849} C_VEL
LIN {X 0,Y 240.667,Z 922.813,A -85,B 0,C 180,E1 11853.341,E2 11853.341} C_VEL
LIN {X 0,Y 249.555,Z 918.083,A -85,B 0,C 180,E1 11849.147,E2 11849.147} C_VEL
LIN {X 0,Y 259.426,Z 911.765,A -85,B 0,C 180,E1 11845.49,E2 11845.49} C_VEL
LIN {X 0,Y 270.676,Z 903.674,A -85,B 0,C 180,E1 11842.18,E2 11842.18} C_VEL
LIN {X 0,Y 275.009,Z 900.4,A -85,B 0,C 180,E1 11841.084,E2 11841.084} C_VEL
LIN {X 0,Y 261.247,Z 913.361,A -85,B 0,C 180,E1 11837.946,E2 11837.946} C_VEL
LIN {X 0,Y 257.205,Z 917.379,A -85,B 0,C 180,E1 11836.811,E2 11836.811} C_VEL
